# B&R Automation Studio project PickNPlaceD5Demo
Automation Studio 6.0.2.177; technology packages: mappCockpit 6.0.0, mappMotion 6.2.0, mappView 6.0.0, OpcUaCs 6.0.0

## Configuration Config1

### Task classes (Cpu.sw)
```
Cyclic#1 (cycle 2000 us, tolerance 0 us):
  APP_ConOut <- Conveyor.APP_ConveyorOut.prg
  APP_ConIn <- Conveyor.APP_ConveyorIn.prg
  APP_Robot1 <- Robots.Robot1.APP_Robot1.prg
DataObjects: McAcpSys, Arnc0sys, Acp10sys
NcDataObjects: mcdrivelog, gmcipuc, gmciplog, gmcipfub, gmcipfun, gmciplsm, gmciplbr, gmcipmxd, gmcipvar, gmcipsys, gmcipiec, gmcipesm, gmcipusm, gmcipcsm, gmcipui, gmcipubr, gmcipcbr, gmcipcfg, gmcipus, gmcipmx, Cam
Binaries: udbdef, TCData, mvLoader, arsvcreg, arflatprv, mCoWebSc, McAcpDrv, McAcpSim, McProfGen, McMechSys, arcoal, ashwac, arconfig, asfw, ashwd, iomap, User, Role, sysconf, TraceConfi, Settings, Config_1, Hierarchy, Config, AxisAx_1, Config_9, ComRobot, Config_7, Config_8, Config_6, ToolX20, AxesAxX21, GRobot1, GFRobot1, ARobot1, ComRobot1, WorkRobot1, GRobot2, MRobot1, GFRobot2, FeatX21, TrkDevX21, TrkDevConv, AxisAxX25, MecX20, AxesAxX20, WorkX20, FeatX20, DeltaX20, ComFeatX20, DeltaX21, TrkDevX20, vccddbox, vcfile, vccbtn, vcpdvnc, arialbd, vcmgr, vctcal, vcgclass, vcctext, vccnum, vcfntttf, vcdsloc, vccstr, arial, Visu03, vccshape, vcalarm, Visu01, vccdt, vccscale, vcchtml, vcchspot, vccbmp, vccpopup, vcshared, vcxml, vccurl, vcrt, vccslider, Visu02, vcnet, vcclbox, vcbclass, vcdsint, vcpdsw, vccovl, vccline, TCLang, visvc, vccdbox, vcpfar00, vcpfmtcx, vcpfapc, GrpMaster, Users, UsersLogin, TC, Files, DiagWebXs, AlmMaster, AlmHisMain, AlmMain, GrpVMaster, AlmVMaster, CfgPureVir, AxisPS, AxisAxXX1, AxisAxXX2, AxisMaster, MDevXX1, AxVMaster, GrpDevXX1, AlmDevXX1, GrPDevXX4, AlmDevXX4, GrPDevX10, AlmDevX10, AlmDevX20, GrpDevX20, AlmDevX21, GrpDevX21, AlmMBelts, GrpMBelts, AlmDevXX6, GrpDevXX6, AxesVAxX20, vcpfx20, AxisMBelts, MasMBelts, MBeltsPt, AxesVAxX25, AxesAxX10, AxesAxX25, WorkX10, CncXX6, MecX10, AxesVAxX10, DeltaX10, FeatXX6, FeatX10, ToolX10, ToolXX6, MecXX6, MotMaster, MotVMaster, vcctrend, MotDevX10, GrPDevXX3, AlmDevXX3, MotDevXX3, GrPDevXX2, MotDevXX1, AlmDevXX2, MotDevXX2, vcpkat, arnc0cfg, Sdc10map, Arnc0map, Sdc10map1, Sdc10map2, MotDevX20, MotDevX11, MotDevXX9, GrpDevXX9, AlmDevXX9, PML, MotDevXX6, CncDevXX6, MotDevXX7, AlmDevXX7, GrpDevXX7, Robot, AlmDevXX8, GrpDevXX8, MotSim, MotSpindle, MotDevXXA, AlmDevXXA, GrpDevXXA, GrpDevX11, AlmDevX11, OpcUaBasic, User_1, OpcUaMap, AlmHmi, AlmHistHmi, Groups, vccpiech, MotMac, acp10cfg, Acp10map
Libraries: standard, AsBrStr, sys_lib, runtime, AsArSdm, astime, brsystem, FileIO, AsIODiag, DataObj, AsArProf, AsMem, AsIOAcc, AsEPL, ASMcDcs, AsBrMath, visapi, ArTextSys, AsSem, AsIecCon, AsZip, powerlnk, aruser, asusb, ashw, arcert, arssl, aseth, asio, asarlog, vcresman, IecCheck, areventlog, MpRecipe, MpUserX, MpFile, MpAlarmX, MpCom, CoTrace, MpServer, McBase, MpBase, MpAxis, McAcpAx, McPathGen, McPureVAx, McAxGroup, McAxis, McProgInt, McTrkPath, McDS402Ax, MpRobotics, MpCnc, MpTool
```

### Hardware
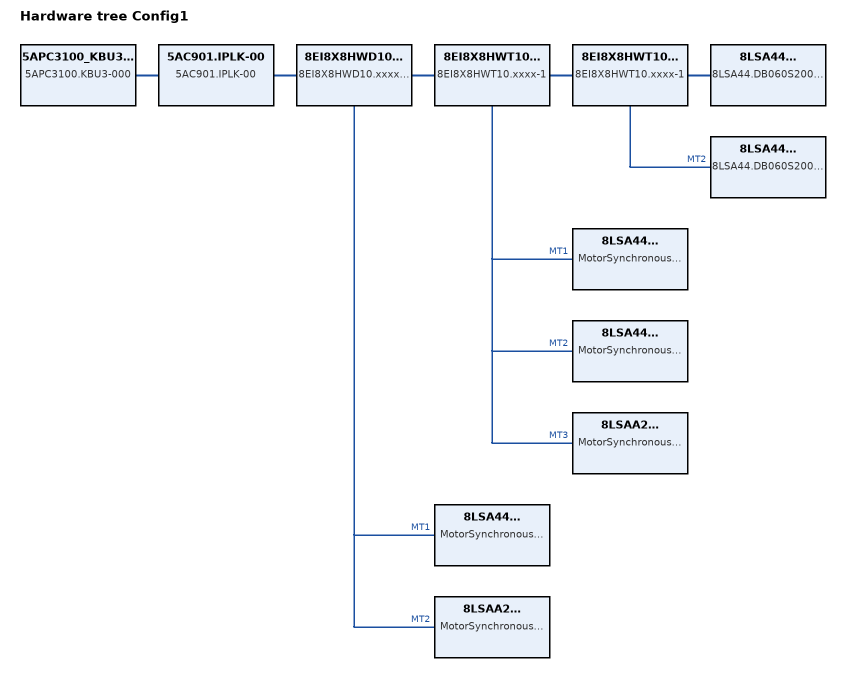
```
5AC901.IPLK-00 : 5AC901.IPLK-00 v2.0.0.0  [SL -> 5APC3100_KBU3_000.SL2]
  Connector IF1:
    DNAConfiguration = manual
    Channel1
    ChannelID1 = McAcpBroadcast
    ChannelType1 = OCTET[96]
5APC3100_KBU3_000 : 5APC3100.KBU3-000 v2.2.7.0
  Connector IF3:
    AssignedOperatingSystem = ARemb
    ActivateDevice = 1
    HostName = apc3100robert
    Mode = Manual
    InternetAddress = 10.43.51.43
    SubnetMask = 255.255.255.0
    Vnc1
    VncKeyMappingFile1 = 
    VncRefreshRate1 = 100
    ActivateSnmp = 2
  Connector IF4:
    AssignedOperatingSystem = ARemb
    ActivateDevice = 1
    HostName = apc3100robert
    Mode = DHCP Server
    InternetAddress = 192.168.20.254
    SubnetMask = 255.255.255.0
    Lease1
    LeaseName1 = Range1
    LeaseStartAddress1 = 192.168.20.100
    LeaseStopAddress1 = 192.168.20.110
    LeaseSubnetMask1 = 255.255.255.0
    Vnc1
    VncTitle1 = VNC
    ActivateSnmp = 2
  Connector IF5:
    AssignedOperatingSystem = ARemb
  Connector IF6:
    AssignedOperatingSystem = ARemb
  Connector IF7:
    AssignedOperatingSystem = ARemb
  Connector IF8:
    AssignedOperatingSystem = ARemb
  ConfigurationID = Template_X20CP1586
  UserPartitionSize = 5
  Simulation = 1
  TimerDeviceType = EPLX2X
  TimerDevice = 5AC901.IPLK-00.IF1
  IdleTaskClass = 4
  TaskClassIdleTime = 4000
  Cyclic1Duration = 2000
  Cyclic1Tolerance = 0
  Cyclic1Stack = 16384
  Cyclic2Duration = 4000
  Cyclic2Tolerance = 0
  Cyclic3Duration = 10000
  Cyclic3Tolerance = 0
  Cyclic4Duration = 20000
  Cyclic4Tolerance = 0
  Cyclic5Duration = 50000
  Cyclic5Tolerance = 0
  Cyclic6Duration = 100000
  Cyclic6Tolerance = 0
  Cyclic7Duration = 200000
  Cyclic7Tolerance = 0
  FileDevice1
  FileDeviceName1 = SceneViewer
  FileDevicePath1 = USER_PATH\..\..\..\..\..\FileDevices\SceneViewer
  FileDevice2
  FileDeviceName2 = CNC_PrgDir
  FileDevicePath2 = USER_PATH\..\..\..\..\..\FileDevices\GCode
  FileDevice3
  FileDeviceName3 = MPLogDir
  FileDevicePath3 = USER_PATH\..\..\..\..\..\FileDevices\Log
  FileDevice4
  FileDeviceName4 = DebugData
  FileDevicePath4 = USER_PATH\..\..\..\..\..\FileDevices\Debug
  EthernetDefaultGateway = 10.43.51.1
  ActivateFtpServer = 1
  FTPProtocol = 2
  FtpUser1
  FtpUsername1 = gmctest
  FtpUserPassword1 = dJg12F/7hd2fGO/QauVo5qNTeUud8LRwkPqca2btE1Q=
  FtpUserSalt1 = iGhlfz5v
  FTPAccessRight1 = 0
  FTPdevice1 = ALL
  ActivateWebServer = 1
  ActivateSdm = 1
8EI8X8HWD10.xxxx-1b_D5r1100R_1 : 8EI8X8HWD10.xxxx-1 v2.3.2.0 (NodeNumber=1)  [PLK1 -> 5AC901.IPLK-00.IF1 [Cable Type=PowerlinkCable, Length=10, Version=1.0.0.3]; PLK2 -> 8EI8X8HWT10.xxxx-1a_D5r1100R_1.PLK1 [Cable Type=PowerlinkCable, Length=10, Version=1.0.0.3]; MT2 -> 8LSAA2.D9045S200-3e_D5r1100R_1.MT]
  DriveConfiguration/Encoder/EncoderX41:
    InterfaceType = EnDat
  DriveConfiguration/Encoder/EncoderX42:
    InterfaceType = EnDat
  DriveConfiguration/Channel[1]/RealAxis:
    AxisReference = gAxisQ3_D5r1100R_1
  DriveConfiguration/Channel[1]/RealAxis/MechanicalElements/Gearbox:
    Input = 10
  DriveConfiguration/Channel[1]/RealAxis/EncoderLink:
    MotorAndPositionEncoder = EncoderX42
  DriveConfiguration/Channel[1]/RealAxis/Controller:
    Mode = PositionControllerWithTorqueFeedForward
  DriveConfiguration/Channel[1]/RealAxis/Controller/Mode/Position:
    ProportionalGain = 1.25
  DriveConfiguration/Channel[1]/RealAxis/Controller/Mode/Speed:
    ProportionalGain = 10.0
  DriveConfiguration/Channel[1]/RealAxis/Controller/Mode:
    FeedForward = CyclicValueFromAxesGroup
  DriveConfiguration/Channel[1]/RealAxis/Homing:
    Mode = Absolute
    RestorePositionVariable = 
  DriveConfiguration/Channel[1]/RealAxis/StopReaction:
    DriveError = CyclicDecelerationFromAxesGroup
  DriveConfiguration/Channel[1]/RealAxis/MovementErrorLimits:
    PositionError = 0.5
  DriveConfiguration/Channel[1]/RealAxis:
    JerkFilter = Used
  DriveConfiguration/Channel[1]/RealAxis/JerkFilter:
    JerkTime = 0.09
  DriveConfiguration/Channel[1]/RealAxis/DigitalInputs/HomingSwitch:
    Source = X8Trigger2
  DriveConfiguration/Channel[2]/RealAxis:
    AxisReference = gAxisQ5_D5r1100R_1
  DriveConfiguration/Channel[2]/RealAxis/MechanicalElements/Gearbox:
    Input = 10
  DriveConfiguration/Channel[2]/RealAxis/Controller:
    Mode = PositionControllerWithTorqueFeedForward
  DriveConfiguration/Channel[2]/RealAxis/Controller/Mode/Position:
    ProportionalGain = 25
  DriveConfiguration/Channel[2]/RealAxis/Controller/Mode/Speed:
    ProportionalGain = 1.25
  DriveConfiguration/Channel[2]/RealAxis/Controller/Mode:
    FeedForward = CyclicValueFromAxesGroup
  DriveConfiguration/Channel[2]/RealAxis/Homing:
    Mode = Absolute
    RestorePositionVariable = 
  DriveConfiguration/Channel[2]/RealAxis/StopReaction:
    DriveError = CyclicDecelerationFromAxesGroup
  DriveConfiguration/Channel[2]/RealAxis/MovementErrorLimits:
    PositionError = 0.5
  DriveConfiguration/Channel[2]/RealAxis:
    JerkFilter = Used
  DriveConfiguration/Channel[2]/RealAxis/JerkFilter:
    JerkTime = 0.09
8EI8X8HWT10.xxxx-1 : 8EI8X8HWT10.xxxx-1 v2.3.2.0 (NodeNumber=3)  [PLK1 -> 8EI8X8HWT10.xxxx-1a_D5r1100R_1.PLK2 [Cable Type=PowerlinkCable, Length=10, Version=1.0.0.3]; MT2 -> 8LSA44.DB060S200-3a.MT]
  DriveConfiguration/Module:
    McAcoposTypeID = AcoposP3TConfig
    ActivateACOPOSSimulationOnPLC = 0
    PowerSupply = AC
  DriveConfiguration/Encoder/EncoderX41:
    InterfaceType = NotUsed
  DriveConfiguration/Encoder/EncoderX42:
    InterfaceType = NotUsed
  DriveConfiguration/Encoder/EncoderX43:
    InterfaceType = NotUsed
  DriveConfiguration/Channel[1]/RealAxis:
    AxisReference = AxConveyorIn
    MechanicalElementsIsInvisible = 0
  DriveConfiguration/Channel[1]/RealAxis/MechanicalElements/Gearbox:
    InputIsReadOnly = 0
    Input = 1
    OutputIsReadOnly = 0
    Output = 1
  DriveConfiguration/Channel[1]/RealAxis/MechanicalElements/RotaryToLinearTransformation:
    ReferenceDistanceIsReadOnly = 0
    ReferenceDistance = 1
  DriveConfiguration/Channel[1]/RealAxis:
    EncoderLink = OneEncoder
  DriveConfiguration/Channel[1]/RealAxis/Controller:
    ModeIsReadOnly = 0
    Mode = PositionController
  DriveConfiguration/Channel[1]/RealAxis/Homing:
    ModeIsReadOnly = 0
    Mode = Direct
    RestorePositionVariable = 
  DriveConfiguration/Channel[1]/RealAxis/StopReaction:
    QuickstopIsReadOnly = 0
    Quickstop = DecelerationLimit
    DriveErrorIsReadOnly = 0
    DriveError = DecelerationLimit
  DriveConfiguration/Channel[1]/RealAxis/MovementErrorLimits:
    PositionError = 1.0
    VelocityErrorMonitoring = Automatic1
  DriveConfiguration/Channel[1]/RealAxis:
    JerkFilterIsReadOnly = 0
    JerkFilter = NotUsed
    ZeroVibrationFilter = NotUsed
  DriveConfiguration/Channel[1]/RealAxis/DigitalInputs/HomingSwitch:
    SourceIsReadOnly = 0
    Source = NotUsed
    Level = High
  DriveConfiguration/Channel[1]/RealAxis/DigitalInputs/PositiveLimitSwitch:
    SourceIsReadOnly = 0
    Source = NotUsed
    Level = High
  DriveConfiguration/Channel[1]/RealAxis/DigitalInputs/NegativeLimitSwitch:
    SourceIsReadOnly = 0
    Source = NotUsed
    Level = High
  DriveConfiguration/Channel[1]/RealAxis/DigitalInputs/Trigger1:
    Source = X8Trigger1
    Level = High
  DriveConfiguration/Channel[1]/RealAxis/DigitalInputs/Trigger2:
    Source = X8Trigger2
    Level = High
  DriveConfiguration/Channel[1]/RealAxis/DigitalInputs/Quickstop:
    Input = Trigger2
  DriveConfiguration/Channel[1]/RealAxis/Simulation:
    SimulationModeOnPLC = SetValueGeneration
    SimulationModeOnACOPOS = NotUsed
  DriveConfiguration/Channel[1]:
    VirtualAxis = NotUsed
    ExternalEncoderAxis = NotUsed
  DriveConfiguration/Channel[2]/RealAxis:
    AxisReference = AxConveyorOut
    MechanicalElementsIsInvisible = 0
  DriveConfiguration/Channel[2]/RealAxis/MechanicalElements/Gearbox:
    InputIsReadOnly = 0
    Input = 1
    OutputIsReadOnly = 0
    Output = 1
  DriveConfiguration/Channel[2]/RealAxis/MechanicalElements/RotaryToLinearTransformation:
    ReferenceDistanceIsReadOnly = 0
    ReferenceDistance = 1
  DriveConfiguration/Channel[2]/RealAxis:
    EncoderLink = OneEncoder
  DriveConfiguration/Channel[2]/RealAxis/Controller:
    ModeIsReadOnly = 0
    Mode = PositionController
  DriveConfiguration/Channel[2]/RealAxis/Homing:
    ModeIsReadOnly = 0
    Mode = Direct
    RestorePositionVariable = 
  DriveConfiguration/Channel[2]/RealAxis/StopReaction:
    QuickstopIsReadOnly = 0
    Quickstop = DecelerationLimit
    DriveErrorIsReadOnly = 0
    DriveError = DecelerationLimit
  DriveConfiguration/Channel[2]/RealAxis/MovementErrorLimits:
    PositionError = 1.0
    VelocityErrorMonitoring = Automatic1
  DriveConfiguration/Channel[2]/RealAxis:
    JerkFilterIsReadOnly = 0
    JerkFilter = NotUsed
    ZeroVibrationFilter = NotUsed
  DriveConfiguration/Channel[2]/RealAxis/DigitalInputs/HomingSwitch:
    SourceIsReadOnly = 0
    Source = NotUsed
    Level = High
  DriveConfiguration/Channel[2]/RealAxis/DigitalInputs/PositiveLimitSwitch:
    SourceIsReadOnly = 0
    Source = NotUsed
    Level = High
  DriveConfiguration/Channel[2]/RealAxis/DigitalInputs/NegativeLimitSwitch:
    SourceIsReadOnly = 0
    Source = NotUsed
    Level = High
  DriveConfiguration/Channel[2]/RealAxis/DigitalInputs/Trigger1:
    Source = X8Trigger1
    Level = High
  DriveConfiguration/Channel[2]/RealAxis/DigitalInputs/Trigger2:
    Source = X8Trigger2
    Level = High
  DriveConfiguration/Channel[2]/RealAxis/DigitalInputs/Quickstop:
    Input = Trigger2
  DriveConfiguration/Channel[2]/RealAxis/Simulation:
    SimulationModeOnPLC = SetValueGeneration
    SimulationModeOnACOPOS = NotUsed
  DriveConfiguration/Channel[2]/RealAxis/AxisFeatures:
    FeatureRef[1] = AxProfGenJerkLim
  DriveConfiguration/Channel[2]:
    VirtualAxis = NotUsed
    ExternalEncoderAxis = NotUsed
  DriveConfiguration/Channel[3]/RealAxis:
    AxisReference = 
    MechanicalElementsIsInvisible = 0
  DriveConfiguration/Channel[3]/RealAxis/MechanicalElements/Gearbox:
    InputIsReadOnly = 0
    Input = 1
    OutputIsReadOnly = 0
    Output = 1
  DriveConfiguration/Channel[3]/RealAxis/MechanicalElements/RotaryToLinearTransformation:
    ReferenceDistanceIsReadOnly = 0
    ReferenceDistance = 1
  DriveConfiguration/Channel[3]/RealAxis:
    EncoderLink = OneEncoder
  DriveConfiguration/Channel[3]/RealAxis/Controller:
    ModeIsReadOnly = 0
    Mode = PositionController
  DriveConfiguration/Channel[3]/RealAxis/Homing:
    ModeIsReadOnly = 0
    Mode = Direct
    RestorePositionVariable = 
  DriveConfiguration/Channel[3]/RealAxis/StopReaction:
    QuickstopIsReadOnly = 0
    Quickstop = DecelerationLimit
    DriveErrorIsReadOnly = 0
    DriveError = DecelerationLimit
  DriveConfiguration/Channel[3]/RealAxis/MovementErrorLimits:
    PositionError = 1.0
    VelocityErrorMonitoring = Automatic1
  DriveConfiguration/Channel[3]/RealAxis:
    JerkFilterIsReadOnly = 0
    JerkFilter = Used
  DriveConfiguration/Channel[3]/RealAxis/JerkFilter:
    JerkTime = 0.09
  DriveConfiguration/Channel[3]/RealAxis:
    ZeroVibrationFilter = NotUsed
  DriveConfiguration/Channel[3]/RealAxis/DigitalInputs/HomingSwitch:
    SourceIsReadOnly = 0
    Source = NotUsed
    Level = High
  DriveConfiguration/Channel[3]/RealAxis/DigitalInputs/PositiveLimitSwitch:
    SourceIsReadOnly = 0
    Source = NotUsed
    Level = High
  DriveConfiguration/Channel[3]/RealAxis/DigitalInputs/NegativeLimitSwitch:
    SourceIsReadOnly = 0
    Source = NotUsed
    Level = High
  DriveConfiguration/Channel[3]/RealAxis/DigitalInputs/Trigger1:
    Source = X8Trigger1
    Level = High
  DriveConfiguration/Channel[3]/RealAxis/DigitalInputs/Trigger2:
    Source = X8Trigger2
    Level = High
  DriveConfiguration/Channel[3]/RealAxis/DigitalInputs/Quickstop:
    Input = Trigger2
  DriveConfiguration/Channel[3]/RealAxis/Simulation:
    SimulationModeOnPLC = SetValueGeneration
    SimulationModeOnACOPOS = NotUsed
  DriveConfiguration/Channel[3]:
    VirtualAxis = NotUsed
    ExternalEncoderAxis = NotUsed
8EI8X8HWT10.xxxx-1a_D5r1100R_1 : 8EI8X8HWT10.xxxx-1 v2.3.2.0 (NodeNumber=2)  [PLK1 -> 8EI8X8HWD10.xxxx-1b_D5r1100R_1.PLK2 [Cable Type=PowerlinkCable, Length=10, Version=1.0.0.3]; PLK2 -> 8EI8X8HWT10.xxxx-1.PLK1 [Cable Type=PowerlinkCable, Length=10, Version=1.0.0.3]; MT2 -> 8LSA44.DB060S200-3b_D5r1100R_1.MT; MT3 -> 8LSAA2.D9045S200-3d_D5r1100R_1.MT]
  DriveConfiguration/Encoder/EncoderX41:
    InterfaceType = EnDat
  DriveConfiguration/Encoder/EncoderX42:
    InterfaceType = EnDat
  DriveConfiguration/Encoder/EncoderX43:
    InterfaceType = EnDat
  DriveConfiguration/Channel[1]/RealAxis:
    AxisReference = gAxisQ1_D5r1100R_1
  DriveConfiguration/Channel[1]/RealAxis/MechanicalElements/Gearbox:
    Input = 28
  DriveConfiguration/Channel[1]/RealAxis/Controller:
    Mode = PositionControllerWithTorqueFeedForward
  DriveConfiguration/Channel[1]/RealAxis/Controller/Mode/Position:
    ProportionalGain = 25
  DriveConfiguration/Channel[1]/RealAxis/Controller/Mode/Speed:
    ProportionalGain = 10
  DriveConfiguration/Channel[1]/RealAxis/Controller/Mode:
    FeedForward = CyclicValueFromAxesGroup
  DriveConfiguration/Channel[1]/RealAxis/Homing:
    Mode = Absolute
    RestorePositionVariable = 
  DriveConfiguration/Channel[1]/RealAxis/StopReaction:
    DriveError = CyclicDecelerationFromAxesGroup
  DriveConfiguration/Channel[1]/RealAxis/MovementErrorLimits:
    PositionError = 0.5
  DriveConfiguration/Channel[1]/RealAxis:
    JerkFilter = Used
  DriveConfiguration/Channel[1]/RealAxis/JerkFilter:
    JerkTime = 0.09
  DriveConfiguration/Channel[2]/RealAxis:
    AxisReference = gAxisQ2_D5r1100R_1
  DriveConfiguration/Channel[2]/RealAxis/MechanicalElements/Gearbox:
    Input = 28
  DriveConfiguration/Channel[2]/RealAxis/Controller:
    Mode = PositionControllerWithTorqueFeedForward
  DriveConfiguration/Channel[2]/RealAxis/Controller/Mode/Position:
    ProportionalGain = 25
  DriveConfiguration/Channel[2]/RealAxis/Controller/Mode/Speed:
    ProportionalGain = 10
  DriveConfiguration/Channel[2]/RealAxis/Controller/Mode:
    FeedForward = CyclicValueFromAxesGroup
  DriveConfiguration/Channel[2]/RealAxis/Homing:
    Mode = Absolute
    RestorePositionVariable = 
  DriveConfiguration/Channel[2]/RealAxis/StopReaction:
    DriveError = CyclicDecelerationFromAxesGroup
  DriveConfiguration/Channel[2]/RealAxis/MovementErrorLimits:
    PositionError = 0.5
  DriveConfiguration/Channel[2]/RealAxis:
    JerkFilter = Used
  DriveConfiguration/Channel[2]/RealAxis/JerkFilter:
    JerkTime = 0.09
  DriveConfiguration/Channel[3]/RealAxis:
    AxisReference = gAxisQ4_D5r1100R_1
  DriveConfiguration/Channel[3]/RealAxis/MechanicalElements/Gearbox:
    Input = 10
  DriveConfiguration/Channel[3]/RealAxis/Controller:
    Mode = PositionControllerWithTorqueFeedForward
  DriveConfiguration/Channel[3]/RealAxis/Controller/Mode/Position:
    ProportionalGain = 350
  DriveConfiguration/Channel[3]/RealAxis/Controller/Mode/Speed:
    ProportionalGain = 0.75
  DriveConfiguration/Channel[3]/RealAxis/Controller/Mode:
    FeedForward = CyclicValueFromAxesGroup
  DriveConfiguration/Channel[3]/RealAxis/Homing:
    Mode = Absolute
    RestorePositionVariable = 
  DriveConfiguration/Channel[3]/RealAxis/StopReaction:
    DriveError = CyclicDecelerationFromAxesGroup
  DriveConfiguration/Channel[3]/RealAxis/MovementErrorLimits:
    PositionError = 0.5
  DriveConfiguration/Channel[3]/RealAxis:
    JerkFilter = Used
  DriveConfiguration/Channel[3]/RealAxis/JerkFilter:
    JerkTime = 0.09
8LSA44.DB060S200-3 : 8LSA44.DB060S200-3 v2.2.0.2  [MT -> 8EI8X8HWT10.xxxx-1.MT1]
  M1/MotorParameters:
    MOTOR_AMB_TEMP_RATED = 40
  M1/MotorParameters/TemperatureSensor:
    MOTOR_TEMPSENS_LIM = 130
8LSA44.DB060S200-3a : 8LSA44.DB060S200-3 v2.2.0.2  [MT -> 8EI8X8HWT10.xxxx-1.MT2]
  M1/MotorParameters:
    MOTOR_AMB_TEMP_RATED = 40
  M1/MotorParameters/TemperatureSensor:
    MOTOR_TEMPSENS_LIM = 130
8LSA44.DB060S200-3a_D5r1100R_1 : MotorSynchronous_any v2.2.1.0  [MT -> 8EI8X8HWT10.xxxx-1a_D5r1100R_1.MT1]
  M1IsInvisible = 0
  TypeIsReadOnly = 0
  M1/MotorParameters:
    MOTOR_POLEPAIRS = 5
    MOTOR_SPEED_RATED = 6000
    MOTOR_SPEED_MAX = 12000
    MOTOR_VOLTAGE_RATED = 400
    MOTOR_CURR_RATED = 3.7
    MOTOR_CURR_STALL = 7.4
    MOTOR_CURR_MAX = 43.8
    MOTOR_TORQ_RATED = 3
    MOTOR_TORQ_STALL = 6
    MOTOR_TORQ_MAX = 22.8
    MOTOR_VOLTAGE_CONST = 49.22
    MOTOR_TORQ_CONST = 0.81
    MOTOR_STATOR_RESISTANCE = 0.862
    MOTOR_STATOR_INDUCTANCE = 6.2
    MOTOR_INERTIA = 2.73
    MOTOR_AMB_TEMP_RATED = 40
    VoltageLimitation = Used
  M1/MotorParameters/VoltageLimitation:
    MOTOR_UDC_MAX = 1000
  M1/MotorParameters/EncoderMounting:
    Angle = StoredOnEncoder
  M1/MotorParameters/TemperatureSensor:
    MOTOR_TEMPSENS_LIM = 130
    TemperatureSensorInterface = EncoderConnectorDigital
    MOTOR_TEMPSENS_PAR1 = 30
    MOTOR_TEMPSENS_PAR2 = 254
    MOTOR_TEMPSENS_PAR3 = -29.72
    MOTOR_TEMPSENS_PAR4 = -4.58
    MOTOR_TEMPSENS_PAR5 = 20.33
    MOTOR_TEMPSENS_PAR6 = 45.18
    MOTOR_TEMPSENS_PAR7 = 69.96
    MOTOR_TEMPSENS_PAR8 = 94.71
    MOTOR_TEMPSENS_PAR9 = 119.6
    MOTOR_TEMPSENS_PAR10 = 149.11
  M1/MotorParameters/TemperatureModel:
    MOTOR_WIND_TEMP_MAX = 110
  M1/MotorParameters/TemperatureModel/Calculation:
    MOTOR_WIND_CROSS_SECT = 0.985
    PIDENT_THERM_TRIP_TIME = 
    MOTOR_TAU_THERM = 1800
  M1:
    Brake = Used
  M1/Brake:
    MOTOR_BRAKE_CURR_RATED = 0.83
    MOTOR_BRAKE_TORQ_RATED = 8
    MOTOR_BRAKE_ON_TIME = 0.038
    MOTOR_BRAKE_OFF_TIME = 0.055
    MOTOR_BRAKE_INERTIA = 0.69
  M1/Encoder:
    MOTOR_ENCOD_ATTR = 1
    MOTOR_ENCOD_INERTIA = 0.022
    TemperatureSensor = Used
  M1/Encoder/TemperatureSensor:
    MOTOR_ENCOD_TEMP_LIM = 129
  M1:
    Gearbox = UsedWithDynamicTorqueLimitation
  M1/Gearbox/GearRatio:
    InputIsReadOnly = 0
    Input = 28
    OutputIsReadOnly = 0
    Output = 1
  M1/Gearbox:
    MOTORGEAR_SPEED_MAX = 5000
    MOTORGEAR_TORQ_NOM = 126
    MOTORGEAR_TORQ_MAX = 126
    MOTORGEAR_INERTIA = 0.51
    MOTORGEAR_VISC_FRIC = 0.002
    MOTORGEAR_STAT_FRIC = 0.22
8LSA44.DB060S200-3b_D5r1100R_1 : MotorSynchronous_any v2.2.1.0  [MT -> 8EI8X8HWT10.xxxx-1a_D5r1100R_1.MT2]
  M1IsInvisible = 0
  TypeIsReadOnly = 0
  M1/MotorParameters:
    MOTOR_POLEPAIRS = 5
    MOTOR_SPEED_RATED = 6000
    MOTOR_SPEED_MAX = 12000
    MOTOR_VOLTAGE_RATED = 400
    MOTOR_CURR_RATED = 3.7
    MOTOR_CURR_STALL = 7.4
    MOTOR_CURR_MAX = 43.8
    MOTOR_TORQ_RATED = 3
    MOTOR_TORQ_STALL = 6
    MOTOR_TORQ_MAX = 22.8
    MOTOR_VOLTAGE_CONST = 49.22
    MOTOR_TORQ_CONST = 0.81
    MOTOR_STATOR_RESISTANCE = 0.862
    MOTOR_STATOR_INDUCTANCE = 6.2
    MOTOR_INERTIA = 2.73
    MOTOR_AMB_TEMP_RATED = 40
    VoltageLimitation = Used
  M1/MotorParameters/VoltageLimitation:
    MOTOR_UDC_MAX = 1000
  M1/MotorParameters/EncoderMounting:
    Angle = StoredOnEncoder
  M1/MotorParameters/TemperatureSensor:
    MOTOR_TEMPSENS_LIM = 130
    TemperatureSensorInterface = EncoderConnectorDigital
    MOTOR_TEMPSENS_PAR1 = 30
    MOTOR_TEMPSENS_PAR2 = 254
    MOTOR_TEMPSENS_PAR3 = -29.72
    MOTOR_TEMPSENS_PAR4 = -4.58
    MOTOR_TEMPSENS_PAR5 = 20.33
    MOTOR_TEMPSENS_PAR6 = 45.18
    MOTOR_TEMPSENS_PAR7 = 69.96
    MOTOR_TEMPSENS_PAR8 = 94.71
    MOTOR_TEMPSENS_PAR9 = 119.6
    MOTOR_TEMPSENS_PAR10 = 149.11
  M1/MotorParameters/TemperatureModel:
    MOTOR_WIND_TEMP_MAX = 110
  M1/MotorParameters/TemperatureModel/Calculation:
    MOTOR_WIND_CROSS_SECT = 0.985
    PIDENT_THERM_TRIP_TIME = 
    MOTOR_TAU_THERM = 1800
  M1:
    Brake = Used
  M1/Brake:
    MOTOR_BRAKE_CURR_RATED = 0.83
    MOTOR_BRAKE_TORQ_RATED = 8
    MOTOR_BRAKE_ON_TIME = 0.038
    MOTOR_BRAKE_OFF_TIME = 0.055
    MOTOR_BRAKE_INERTIA = 0.69
  M1/Encoder:
    MOTOR_ENCOD_ATTR = 1
    MOTOR_ENCOD_INERTIA = 0.022
    TemperatureSensor = Used
  M1/Encoder/TemperatureSensor:
    MOTOR_ENCOD_TEMP_LIM = 129
  M1:
    Gearbox = UsedWithDynamicTorqueLimitation
  M1/Gearbox/GearRatio:
    InputIsReadOnly = 0
    Input = 28
    OutputIsReadOnly = 0
    Output = 1
  M1/Gearbox:
    MOTORGEAR_SPEED_MAX = 5000
    MOTORGEAR_TORQ_NOM = 126
    MOTORGEAR_TORQ_MAX = 126
    MOTORGEAR_INERTIA = 0.51
    MOTORGEAR_VISC_FRIC = 0.002
    MOTORGEAR_STAT_FRIC = 0.22
8LSA44.DB060S200-3c_D5r1100R_1 : MotorSynchronous_any v2.2.1.0  [MT -> 8EI8X8HWD10.xxxx-1b_D5r1100R_1.MT1]
  M1IsInvisible = 0
  TypeIsReadOnly = 0
  M1/MotorParameters:
    MOTOR_POLEPAIRS = 5
    MOTOR_SPEED_RATED = 6000
    MOTOR_SPEED_MAX = 12000
    MOTOR_VOLTAGE_RATED = 400
    MOTOR_CURR_RATED = 3.7
    MOTOR_CURR_STALL = 7.4
    MOTOR_CURR_MAX = 43.8
    MOTOR_TORQ_RATED = 3
    MOTOR_TORQ_STALL = 6
    MOTOR_TORQ_MAX = 22.8
    MOTOR_VOLTAGE_CONST = 49.22
    MOTOR_TORQ_CONST = 0.81
    MOTOR_STATOR_RESISTANCE = 0.862
    MOTOR_STATOR_INDUCTANCE = 6.2
    MOTOR_INERTIA = 2.73
    MOTOR_AMB_TEMP_RATED = 40
    VoltageLimitation = Used
  M1/MotorParameters/VoltageLimitation:
    MOTOR_UDC_MAX = 1000
  M1/MotorParameters/EncoderMounting:
    Angle = StoredOnEncoder
  M1/MotorParameters/TemperatureSensor:
    MOTOR_TEMPSENS_LIM = 130
    TemperatureSensorInterface = EncoderConnectorDigital
    MOTOR_TEMPSENS_PAR1 = 30
    MOTOR_TEMPSENS_PAR2 = 254
    MOTOR_TEMPSENS_PAR3 = -29.72
    MOTOR_TEMPSENS_PAR4 = -4.58
    MOTOR_TEMPSENS_PAR5 = 20.33
    MOTOR_TEMPSENS_PAR6 = 45.18
    MOTOR_TEMPSENS_PAR7 = 69.96
    MOTOR_TEMPSENS_PAR8 = 94.71
    MOTOR_TEMPSENS_PAR9 = 119.6
    MOTOR_TEMPSENS_PAR10 = 149.11
  M1/MotorParameters/TemperatureModel:
    MOTOR_WIND_TEMP_MAX = 110
  M1/MotorParameters/TemperatureModel/Calculation:
    MOTOR_WIND_CROSS_SECT = 0.985
    PIDENT_THERM_TRIP_TIME = 
    MOTOR_TAU_THERM = 1800
  M1:
    Brake = Used
  M1/Brake:
    MOTOR_BRAKE_CURR_RATED = 0.83
    MOTOR_BRAKE_TORQ_RATED = 8
    MOTOR_BRAKE_ON_TIME = 0.038
    MOTOR_BRAKE_OFF_TIME = 0.055
    MOTOR_BRAKE_INERTIA = 0.69
  M1/Encoder:
    MOTOR_ENCOD_ATTR = 1
    MOTOR_ENCOD_INERTIA = 0.022
    TemperatureSensor = Used
  M1/Encoder/TemperatureSensor:
    MOTOR_ENCOD_TEMP_LIM = 129
  M1:
    Gearbox = UsedWithDynamicTorqueLimitation
  M1/Gearbox/GearRatio:
    InputIsReadOnly = 0
    Input = 28
    OutputIsReadOnly = 0
    Output = 1
  M1/Gearbox:
    MOTORGEAR_SPEED_MAX = 5000
    MOTORGEAR_TORQ_NOM = 126
    MOTORGEAR_TORQ_MAX = 126
    MOTORGEAR_INERTIA = 0.51
    MOTORGEAR_VISC_FRIC = 0.002
    MOTORGEAR_STAT_FRIC = 0.22
8LSAA2.D9045S200-3d_D5r1100R_1 : MotorSynchronous_any v2.2.1.0  [MT -> 8EI8X8HWT10.xxxx-1a_D5r1100R_1.MT3]
  M1IsInvisible = 0
  TypeIsReadOnly = 0
  M1/MotorParameters:
    MOTOR_POLEPAIRS = 5
    MOTOR_SPEED_RATED = 4500
    MOTOR_SPEED_MAX = 7000
    MOTOR_VOLTAGE_RATED = 400
    MOTOR_CURR_RATED = 1.31
    MOTOR_CURR_STALL = 1.42
    MOTOR_CURR_MAX = 6
    MOTOR_TORQ_RATED = 1.27
    MOTOR_TORQ_STALL = 1.4
    MOTOR_TORQ_MAX = 4.5
    MOTOR_VOLTAGE_CONST = 58.64
    MOTOR_TORQ_CONST = 0.97
    MOTOR_STATOR_RESISTANCE = 13.9
    MOTOR_STATOR_INDUCTANCE = 27
    MOTOR_INERTIA = 0.38
    MOTOR_AMB_TEMP_RATED = 40
    VoltageLimitation = Used
  M1/MotorParameters/VoltageLimitation:
    MOTOR_UDC_MAX = 1000
  M1/MotorParameters/EncoderMounting:
    Angle = StoredOnEncoder
  M1/MotorParameters/TemperatureSensor:
    MOTOR_TEMPSENS_LIM = 130
    TemperatureSensorInterface = EncoderConnectorDigital
    MOTOR_TEMPSENS_PAR1 = 30
    MOTOR_TEMPSENS_PAR2 = 254
    MOTOR_TEMPSENS_PAR3 = -29.72
    MOTOR_TEMPSENS_PAR4 = -4.58
    MOTOR_TEMPSENS_PAR5 = 20.33
    MOTOR_TEMPSENS_PAR6 = 45.18
    MOTOR_TEMPSENS_PAR7 = 69.96
    MOTOR_TEMPSENS_PAR8 = 94.71
    MOTOR_TEMPSENS_PAR9 = 119.6
    MOTOR_TEMPSENS_PAR10 = 149.11
  M1/MotorParameters/TemperatureModel:
    MOTOR_WIND_TEMP_MAX = 110
  M1/MotorParameters/TemperatureModel/Calculation:
    MOTOR_WIND_CROSS_SECT = 0.126
    MOTOR_TAU_THERM = 1860
  M1:
    Brake = Used
  M1/Brake:
    MOTOR_BRAKE_CURR_RATED = 0.56
    MOTOR_BRAKE_TORQ_RATED = 3.2
    MOTOR_BRAKE_ON_TIME = 0.01
    MOTOR_BRAKE_OFF_TIME = 0.06
    MOTOR_BRAKE_INERTIA = 0.38
  M1/Encoder:
    MOTOR_ENCOD_ATTR = 1
    MOTOR_ENCOD_INERTIA = 0.004
    TemperatureSensor = Used
  M1/Encoder/TemperatureSensor:
    MOTOR_ENCOD_TEMP_LIM = 124
  M1:
    Gearbox = UsedWithDynamicTorqueLimitation
  M1/Gearbox/GearRatio:
    InputIsReadOnly = 0
    Input = 10
    OutputIsReadOnly = 0
    Output = 1
  M1/Gearbox:
    MOTORGEAR_SPEED_MAX = 7500
    MOTORGEAR_TORQ_NOM = 7
    MOTORGEAR_TORQ_MAX = 7
    MOTORGEAR_INERTIA = 0.16
    MOTORGEAR_VISC_FRIC = 0.01
    MOTORGEAR_STAT_FRIC = 0.1
8LSAA2.D9045S200-3e_D5r1100R_1 : MotorSynchronous_any v2.2.1.0  [MT -> 8EI8X8HWD10.xxxx-1b_D5r1100R_1.MT2]
  M1IsInvisible = 0
  TypeIsReadOnly = 0
  M1/MotorParameters:
    MOTOR_POLEPAIRS = 5
    MOTOR_SPEED_RATED = 4500
    MOTOR_SPEED_MAX = 7000
    MOTOR_VOLTAGE_RATED = 400
    MOTOR_CURR_RATED = 1.31
    MOTOR_CURR_STALL = 1.42
    MOTOR_CURR_MAX = 6
    MOTOR_TORQ_RATED = 1.27
    MOTOR_TORQ_STALL = 1.4
    MOTOR_TORQ_MAX = 4.5
    MOTOR_VOLTAGE_CONST = 58.64
    MOTOR_TORQ_CONST = 0.97
    MOTOR_STATOR_RESISTANCE = 13.9
    MOTOR_STATOR_INDUCTANCE = 27
    MOTOR_INERTIA = 0.38
    MOTOR_AMB_TEMP_RATED = 40
    VoltageLimitation = Used
  M1/MotorParameters/VoltageLimitation:
    MOTOR_UDC_MAX = 1000
  M1/MotorParameters/EncoderMounting:
    Angle = StoredOnEncoder
  M1/MotorParameters/TemperatureSensor:
    MOTOR_TEMPSENS_LIM = 130
    TemperatureSensorInterface = EncoderConnectorDigital
    MOTOR_TEMPSENS_PAR1 = 30
    MOTOR_TEMPSENS_PAR2 = 254
    MOTOR_TEMPSENS_PAR3 = -29.72
    MOTOR_TEMPSENS_PAR4 = -4.58
    MOTOR_TEMPSENS_PAR5 = 20.33
    MOTOR_TEMPSENS_PAR6 = 45.18
    MOTOR_TEMPSENS_PAR7 = 69.96
    MOTOR_TEMPSENS_PAR8 = 94.71
    MOTOR_TEMPSENS_PAR9 = 119.6
    MOTOR_TEMPSENS_PAR10 = 149.11
  M1/MotorParameters/TemperatureModel:
    MOTOR_WIND_TEMP_MAX = 110
  M1/MotorParameters/TemperatureModel/Calculation:
    MOTOR_WIND_CROSS_SECT = 0.126
    MOTOR_TAU_THERM = 1860
  M1:
    Brake = Used
  M1/Brake:
    MOTOR_BRAKE_CURR_RATED = 0.56
    MOTOR_BRAKE_TORQ_RATED = 3.2
    MOTOR_BRAKE_ON_TIME = 0.01
    MOTOR_BRAKE_OFF_TIME = 0.06
    MOTOR_BRAKE_INERTIA = 0.38
  M1/Encoder:
    MOTOR_ENCOD_ATTR = 1
    MOTOR_ENCOD_INERTIA = 0.004
    TemperatureSensor = Used
  M1/Encoder/TemperatureSensor:
    MOTOR_ENCOD_TEMP_LIM = 124
  M1:
    Gearbox = UsedWithDynamicTorqueLimitation
  M1/Gearbox/GearRatio:
    InputIsReadOnly = 0
    Input = 10
    OutputIsReadOnly = 0
    Output = 1
  M1/Gearbox:
    MOTORGEAR_SPEED_MAX = 7500
    MOTORGEAR_TORQ_NOM = 7
    MOTORGEAR_TORQ_MAX = 7
    MOTORGEAR_INERTIA = 0.16
    MOTORGEAR_VISC_FRIC = 0.01
    MOTORGEAR_STAT_FRIC = 0.1
```

### Config_10.dynpartable - 5APC3100_KBU3_000/mappMotion/Codian_D5r1100R_1/Config_10.dynpartable
```
Element ProductLoad_2 (Type=dynpartable)
  Row[1]:
    Value = 1.0
    Unit = kg
    Description = Mass
  Row[2]:
    Index = 1
    Unit = m
    Description = Center of gravity - X direction
  Row[3]:
    Index = 2
    Unit = m
    Description = Center of gravity - Y direction
  Row[4]:
    Index = 3
    Unit = m
    Description = Center of gravity - Z direction
  Row[5]:
    Index = 4
    Unit = kg m^2
    Description = Moment of inertia about X
  Row[6]:
    Index = 5
    Unit = kg m^2
    Description = Moment of inertia about Y
  Row[7]:
    Index = 6
    Unit = kg m^2
    Description = Moment of inertia about Z
  Row[8]:
    Index = 1000
    Value = 1
    Unit = 
    Description = 0 (toolDynPar), 1 (productLoadPar)
```

### Config_11.tool - 5APC3100_KBU3_000/mappMotion/Codian_D5r1100R_1/Config_11.tool
```
Element Tool_1 (Type=tool)
```

### Config_4.dynpartable - 5APC3100_KBU3_000/mappMotion/Codian_D5r1100R_1/Config_4.dynpartable
```
Element ProductLoad_1 (Type=dynpartable)
  Row[1]:
    Value = 0.5
    Unit = kg
    Description = Mass
  Row[2]:
    Index = 1
    Unit = m
    Description = Center of gravity - X direction
  Row[3]:
    Index = 2
    Unit = m
    Description = Center of gravity - Y direction
  Row[4]:
    Index = 3
    Unit = m
    Description = Center of gravity - Z direction
  Row[5]:
    Index = 4
    Unit = kg m^2
    Description = Moment of inertia about X
  Row[6]:
    Index = 5
    Unit = kg m^2
    Description = Moment of inertia about Y
  Row[7]:
    Index = 6
    Unit = kg m^2
    Description = Moment of inertia about Z
  Row[8]:
    Index = 1000
    Value = 1
    Unit = 
    Description = 0 (toolDynPar), 1 (productLoadPar)
```

### Config_5.tooltable - 5APC3100_KBU3_000/mappMotion/Codian_D5r1100R_1/Config_5.tooltable
```
Element ToolTable_1 (Type=tooltable)
  Row[1]:
    Index = 3
    ToolDataRef = Tool_1
    ToolDynParDataRef = 
  Row[2]:
    ToolDynParDataRef = ProductLoad_1
  Row[3]:
    Index = 2
    ToolDynParDataRef = ProductLoad_2
```

### Config_6.axesgroup - 5APC3100_KBU3_000/mappMotion/Codian_D5r1100R_1/Config_6.axesgroup
```
Element gAxesGroup_D5r1100R_1 (Type=axesgroup)
  Type = PathGenAxesGroup
    ProcessingTaskClass = 1
    PhysicalAxes:
      JointAxes:
        JointAxis[1]:
          AxisRef = gAxisQ1_D5r1100R_1
        JointAxis[2]:
          AxisRef = gAxisQ2_D5r1100R_1
        JointAxis[3]:
          AxisRef = gAxisQ3_D5r1100R_1
        JointAxis[4]:
          Name = QC
          AxisRef = gAxisQ4_D5r1100R_1
        JointAxis[5]:
          Name = QA
          AxisRef = gAxisQ5_D5r1100R_1
    MechanicalSystem:
      MechSysRef = MechSys_D5r1100R_1
    BasicSettings:
      GeometryPlanning:
        MaxTangentialTransitionDeviation = 0.05
      TrajectoryPlanning:
        LimitCheckResolution:
          Time = 0.005
        BufferTime:
          Time = 0.05
      Miscellaneous:
        TimeStretchOverride:
          JerkSuppression = Basic
            AdaptationTime = 0.3
    StopReaction:
      AxisError:
        AxisReactionIsReadOnly = 1
        AxisReaction = DynamicStop
          ModeIsReadOnly = 1
    AxesGroupFeatures:
      FeatureRef[1] = Feature_Programs_D5r1100R_1
      FeatureRef[2] = Feature_FrameHierachy
      FeatureRef[3] = Feature_InterpreterLog
      FeatureRef[4] = Feature_MFunctions
      FeatureRef[5] = Feature_Monitoring
      FeatureRef[6] = Feature_PathDefRobot
      FeatureRef[7] = Feature_TrackingRobot
      FeatureRef[8] = Feature_WorkspaceMonitoring
      FeatureRef[9] = Feature_Signaling
      FeatureRef[10] = Feature_Tool
```

### Config_7.axis - 5APC3100_KBU3_000/mappMotion/Codian_D5r1100R_1/Config_7.axis
```
Element gAxisQ1_D5r1100R_1 (Type=axis)
  BaseTypeIsReadOnly = 0
  BaseType = RotaryBounded
    MeasurementUnitIsReadOnly = 1
    MeasurementUnit = 17476
    MeasurementResolutionIsReadOnly = 1
    MeasurementResolution = 0.001
    CountDirectionIsReadOnly = 1
    CountDirection = Inverse
  MovementLimitsIsReadOnly = 0
  MovementLimits = InternalForPathControlledAxis
    Position:
      LowerLimitMin = -47
      UpperLimitMax = 99.5
      LowerLimit = -47
      UpperLimit = 99.5
    VelocityIsReadOnly = 0
    Velocity:
      VelocityMax = 3.4E38
      Velocity = 1160
    AccelerationIsReadOnly = 0
    Acceleration:
      AccelerationMax = 3.4E38
      Acceleration = 35000
    DecelerationIsReadOnly = 0
    Deceleration:
      DecelerationMax = 3.4E38
      Deceleration = 35000
    JerkIsReadOnly = 0
    Jerk = Advanced
      JerkAccelerationPositiveMin = 0
      JerkAccelerationPositiveMax = 3.4E38
      JerkAccelerationPositive = 1500000
      JerkAccelerationNegativeMin = 0
      JerkAccelerationNegativeMax = 3.4E38
      JerkAccelerationNegative = 1500000
      JerkDecelerationPositiveMin = 0
      JerkDecelerationPositiveMax = 3.4E38
      JerkDecelerationPositive = 1500000
      JerkDecelerationNegativeMin = 0
      JerkDecelerationNegativeMax = 3.4E38
      JerkDecelerationNegative = 1500000
    TorqueIsInvisible = 0
    TorqueIsReadOnly = 0
    Torque = Basic
      TorqueMax = 3.4E38
      Torque = 11
  Alarms = None
Element gAxisQ2_D5r1100R_1 (Type=axis)
  BaseTypeIsReadOnly = 0
  BaseType = RotaryBounded
    MeasurementUnitIsReadOnly = 1
    MeasurementUnit = 17476
    MeasurementResolutionIsReadOnly = 1
    MeasurementResolution = 0.001
    CountDirectionIsReadOnly = 1
    CountDirection = Inverse
  MovementLimitsIsReadOnly = 0
  MovementLimits = InternalForPathControlledAxis
    Position:
      LowerLimitMin = -47
      UpperLimitMax = 99.5
      LowerLimit = -47
      UpperLimit = 99.5
    VelocityIsReadOnly = 0
    Velocity:
      VelocityMax = 3.4E38
      Velocity = 1160
    AccelerationIsReadOnly = 0
    Acceleration:
      AccelerationMax = 3.4E38
      Acceleration = 35000
    DecelerationIsReadOnly = 0
    Deceleration:
      DecelerationMax = 3.4E38
      Deceleration = 35000
    JerkIsReadOnly = 0
    Jerk = Advanced
      JerkAccelerationPositiveMin = 0
      JerkAccelerationPositiveMax = 3.4E38
      JerkAccelerationPositive = 1500000
      JerkAccelerationNegativeMin = 0
      JerkAccelerationNegativeMax = 3.4E38
      JerkAccelerationNegative = 1500000
      JerkDecelerationPositiveMin = 0
      JerkDecelerationPositiveMax = 3.4E38
      JerkDecelerationPositive = 1500000
      JerkDecelerationNegativeMin = 0
      JerkDecelerationNegativeMax = 3.4E38
      JerkDecelerationNegative = 1500000
    TorqueIsInvisible = 0
    TorqueIsReadOnly = 0
    Torque = Basic
      TorqueMax = 3.4E38
      Torque = 11
  Alarms = None
Element gAxisQ3_D5r1100R_1 (Type=axis)
  BaseTypeIsReadOnly = 0
  BaseType = RotaryBounded
    MeasurementUnitIsReadOnly = 1
    MeasurementUnit = 17476
    MeasurementResolutionIsReadOnly = 1
    MeasurementResolution = 0.001
    CountDirectionIsReadOnly = 1
    CountDirection = Inverse
  MovementLimitsIsReadOnly = 0
  MovementLimits = InternalForPathControlledAxis
    Position:
      LowerLimitMin = -47
      UpperLimitMax = 99.5
      LowerLimit = -47
      UpperLimit = 99.5
    VelocityIsReadOnly = 0
    Velocity:
      VelocityMax = 3.4E38
      Velocity = 1160
    AccelerationIsReadOnly = 0
    Acceleration:
      AccelerationMax = 3.4E38
      Acceleration = 35000
    DecelerationIsReadOnly = 0
    Deceleration:
      DecelerationMax = 3.4E38
      Deceleration = 35000
    JerkIsReadOnly = 0
    Jerk = Advanced
      JerkAccelerationPositiveMin = 0
      JerkAccelerationPositiveMax = 3.4E38
      JerkAccelerationPositive = 1500000
      JerkAccelerationNegativeMin = 0
      JerkAccelerationNegativeMax = 3.4E38
      JerkAccelerationNegative = 1500000
      JerkDecelerationPositiveMin = 0
      JerkDecelerationPositiveMax = 3.4E38
      JerkDecelerationPositive = 1500000
      JerkDecelerationNegativeMin = 0
      JerkDecelerationNegativeMax = 3.4E38
      JerkDecelerationNegative = 1500000
    TorqueIsInvisible = 0
    TorqueIsReadOnly = 0
    Torque = Basic
      TorqueMax = 3.4E38
      Torque = 11
  Alarms = None
Element gAxisQ4_D5r1100R_1 (Type=axis)
  BaseTypeIsReadOnly = 0
  BaseType = Rotary
    MeasurementUnitIsReadOnly = 1
    MeasurementUnit = 17476
    MeasurementResolutionIsReadOnly = 1
    MeasurementResolution = 0.001
    CountDirectionIsReadOnly = 1
    CountDirection = Standard
  MovementLimitsIsReadOnly = 0
  MovementLimits = InternalForPathControlledAxis
    Position:
      LowerLimitMin = -1000.0
      UpperLimitMax = 1000.0
      LowerLimit = -1000.0
      UpperLimit = 1000.0
    VelocityIsReadOnly = 0
    Velocity:
      VelocityMax = 3.4E38
      Velocity = 3600
    AccelerationIsReadOnly = 0
    Acceleration:
      AccelerationMax = 3.4E38
      Acceleration = 100000
    DecelerationIsReadOnly = 0
    Deceleration:
      DecelerationMax = 3.4E38
      Deceleration = 100000
    JerkIsReadOnly = 0
    Jerk = Advanced
      JerkAccelerationPositiveMin = 0
      JerkAccelerationPositiveMax = 3.4E38
      JerkAccelerationPositive = 6000000
      JerkAccelerationNegativeMin = 0
      JerkAccelerationNegativeMax = 3.4E38
      JerkAccelerationNegative = 6000000
      JerkDecelerationPositiveMin = 0
      JerkDecelerationPositiveMax = 3.4E38
      JerkDecelerationPositive = 6000000
      JerkDecelerationNegativeMin = 0
      JerkDecelerationNegativeMax = 3.4E38
      JerkDecelerationNegative = 6000000
    TorqueIsInvisible = 0
    TorqueIsReadOnly = 0
    Torque = Basic
      TorqueMax = 3.4E38
      Torque = 1.2
  Alarms = None
Element gAxisQ5_D5r1100R_1 (Type=axis)
  BaseTypeIsReadOnly = 0
  BaseType = Rotary
    MeasurementUnitIsReadOnly = 1
    MeasurementUnit = 17476
    MeasurementResolutionIsReadOnly = 1
    MeasurementResolution = 0.001
    CountDirectionIsReadOnly = 1
    CountDirection = Standard
  MovementLimitsIsReadOnly = 0
  MovementLimits = InternalForPathControlledAxis
    Position:
      LowerLimitMin = -186.01
      UpperLimitMax = 186.01
      LowerLimit = -186.01
      UpperLimit = 186.01
    VelocityIsReadOnly = 0
    Velocity:
      VelocityMax = 3.4E38
      Velocity = 3300
    AccelerationIsReadOnly = 0
    Acceleration:
      AccelerationMax = 3.4E38
      Acceleration = 100000
    DecelerationIsReadOnly = 0
    Deceleration:
      DecelerationMax = 3.4E38
      Deceleration = 100000
    JerkIsReadOnly = 0
    Jerk = Advanced
      JerkAccelerationPositiveMin = 0
      JerkAccelerationPositiveMax = 3.4E38
      JerkAccelerationPositive = 6000000
      JerkAccelerationNegativeMin = 0
      JerkAccelerationNegativeMax = 3.4E38
      JerkAccelerationNegative = 6000000
      JerkDecelerationPositiveMin = 0
      JerkDecelerationPositiveMax = 3.4E38
      JerkDecelerationPositive = 6000000
      JerkDecelerationNegativeMin = 0
      JerkDecelerationNegativeMax = 3.4E38
      JerkDecelerationNegative = 6000000
    TorqueIsInvisible = 0
    TorqueIsReadOnly = 0
    Torque = Basic
      TorqueMax = 3.4E38
      Torque = 2
  Alarms = None
```

### Config_8.mechanicalsystem - 5APC3100_KBU3_000/mappMotion/Codian_D5r1100R_1/Config_8.mechanicalsystem
```
Element MechSys_D5r1100R_1 (Type=mechanicalsystem)
  TypeIsReadOnly = 1
  Type = Delta
    SubtypeIsReadOnly = 1
    Subtype = 5AxesDeltaA
      SceneViewerObject = Generic
      DescriptionIsReadOnly = 1
      Description = Standard
        Dimensions:
          BasePlatform:
            CenterIsReadOnly = 0
            Center:
              X = 0.0
              Y = 0.0
              Z = 0
            ArmLinkPointIsReadOnly = 0
            Arm1LinkPoint:
              Angle = 0.0
              Radius = 200
              Z = -90
            Arm2LinkPoint:
              Angle = -120.0
              Radius = 200
              Z = -90
            Arm3LinkPoint:
              Angle = -240.0
              Radius = 200
              Z = -90
          Arms:
            ArmIsReadOnly = 0
            Arm1:
              UpperArmLength = 320
              LowerArmLength = 850
            Arm2:
              UpperArmLength = 320
              LowerArmLength = 850
            Arm3:
              UpperArmLength = 320
              LowerArmLength = 850
            LowerArmPairDistance = 104
          EndEffectorPlatform:
            ArmLinkPointIsReadOnly = 0
            Arm1LinkPoint:
              Radius = 66
              Z = 0.0
            Arm2LinkPoint:
              Radius = 66
              Z = 0.0
            Arm3LinkPoint:
              Radius = 66
              Z = 0.0
            TranslationToQCIsReadOnly = 0
            TranslationToQC:
              X = 27.5
              Y = 0.0
              Z = 0.0
            TranslationFromQCToQAIsReadOnly = 0
            TranslationFromQCToQA:
              X = 0.0
              Y = 0.0
              Z = -74.9
            TranslationFromQAToFlangeIsReadOnly = 0
            TranslationFromQAToFlange:
              X = 0.0
              Y = 0.0
              Z = -80
        Offsets:
          JointAxisIsReadOnly = 0
          JointAxis[1] = 0.0
          JointAxis[2] = 0.0
          JointAxis[3] = 0.0
          JointAxis[4] = 0.0
          JointAxis[5] = 0.0
        CountDirections:
          JointAxisIsReadOnly = 0
          JointAxis[1] = Standard
          JointAxis[2] = Standard
          JointAxis[3] = Standard
          JointAxis[4] = Standard
          JointAxis[5] = Standard
      CoordinatesNames = Default
        XCoordinateName = X
        YCoordinateName = Y
        ZCoordinateName = Z
        CCoordinateName = C
        ACoordinateName = A
      TcpOrientation:
        Frames = Used
      WireFrameModelIsReadOnly = 0
      WireFrameModel = Standard
        UpperArm1IsReadOnly = 0
        UpperArm1 = ConnectionLine
          DistanceMin = -1.79769313486231E308
          DistanceMax = 1.79769313486231E308
          Distance = 5
        LowerArm1IsReadOnly = 0
        LowerArm1 = ConnectionLine
          DistanceMin = -1.79769313486231E308
          DistanceMax = 1.79769313486231E308
          Distance = 5
        UpperArm2IsReadOnly = 0
        UpperArm2 = ConnectionLine
          DistanceMin = -1.79769313486231E308
          DistanceMax = 1.79769313486231E308
          Distance = 5
        LowerArm2IsReadOnly = 0
        LowerArm2 = ConnectionLine
          DistanceMin = -1.79769313486231E308
          DistanceMax = 1.79769313486231E308
          Distance = 5
        UpperArm3IsReadOnly = 0
        UpperArm3 = ConnectionLine
          DistanceMin = -1.79769313486231E308
          DistanceMax = 1.79769313486231E308
          Distance = 5
        LowerArm3IsReadOnly = 0
        LowerArm3 = ConnectionLine
          DistanceMin = -1.79769313486231E308
          DistanceMax = 1.79769313486231E308
          Distance = 5
        EndEffectorPlatformToQCIsReadOnly = 0
        EndEffectorPlatformToQC = ConnectionLine
          DistanceMin = -1.79769313486231E308
          DistanceMax = 1.79769313486231E308
          Distance = 0.0
        QCToQAIsReadOnly = 0
        QCToQA = ConnectionLine
          DistanceMin = -1.79769313486231E308
          DistanceMax = 1.79769313486231E308
          Distance = 0.0
        QAToFlangeIsReadOnly = 0
        QAToFlange = ConnectionLine
          DistanceMin = -1.79769313486231E308
          DistanceMax = 1.79769313486231E308
          Distance = 0.0
        FlangeToTcp = NotUsed
      DynamicModelIsReadOnly = 0
      DynamicModel = DynParTable
        TableRef
      InternalDynamicModelIsReadOnly = 1
      InternalDynamicModel = Used
        TypeIsReadOnly = 1
        Type = D5-1100-S026-R100
        Row[1]:
          Index = 0
          Value = 3
          Unit = 
          Description = type of robot dyn par model
        Row[2]:
          Index = 1
          Value = 1.017
          Unit = kg
          Description = m1
        Row[3]:
          Index = 2
          Value = 0.1042425
          Unit = kgm
          Description = m1*rc1x
        Row[4]:
          Index = 3
          Value = 0
          Unit = kgm
          Description = m1*rc1y
        Row[5]:
          Index = 4
          Value = 0.0044748
          Unit = kgm
          Description = m1*rc1z
        Row[6]:
          Index = 5
          Value = 0
          Unit = kgm^2
          Description = m1*rc1x*rc1y
        Row[7]:
          Index = 6
          Value = 0
          Unit = kgm^2
          Description = m1*rc1y*rc1z
        Row[8]:
          Index = 7
          Value = 0.000458667
          Unit = kgm^2
          Description = m1*rc1x*rc1z
        Row[9]:
          Index = 8
          Value = 0.01068485625
          Unit = kgm^2
          Description = m1*rc1x^2
        Row[10]:
          Index = 9
          Value = 0
          Unit = kgm^2
          Description = m1*rc1y^2
        Row[11]:
          Index = 10
          Value = 0.00001968912
          Unit = kgm^2
          Description = m1*rc1z^2
        Row[12]:
          Index = 11
          Value = 0
          Unit = kgm^2
          Description = Jxx1
        Row[13]:
          Index = 12
          Value = 0.0129
          Unit = kgm^2
          Description = Jyy1
        Row[14]:
          Index = 13
          Value = 0
          Unit = kgm^2
          Description = Jzz1
        Row[15]:
          Index = 14
          Value = 1.017
          Unit = kg
          Description = m2
        Row[16]:
          Index = 15
          Value = 0.1042425
          Unit = kgm
          Description = m2*rc2x
        Row[17]:
          Index = 16
          Value = 0
          Unit = kgm
          Description = m2*rc2y
        Row[18]:
          Index = 17
          Value = 0.0044748
          Unit = kgm
          Description = m2*rc2z
        Row[19]:
          Index = 18
          Value = 0
          Unit = kgm^2
          Description = m2*rc2x*rc2y
        Row[20]:
          Index = 19
          Value = 0
          Unit = kgm^2
          Description = m2*rc2y*rc2z
        Row[21]:
          Index = 20
          Value = 0.000458667
          Unit = kgm^2
          Description = m2*rc2x*rc2z
        Row[22]:
          Index = 21
          Value = 0.01068485625
          Unit = kgm^2
          Description = m2*rc2x^2
        Row[23]:
          Index = 22
          Value = 0
          Unit = kgm^2
          Description = m2*rc2y^2
        Row[24]:
          Index = 23
          Value = 0.00001968912
          Unit = kgm^2
          Description = m2*rc2z^2
        Row[25]:
          Index = 24
          Value = 0
          Unit = kgm^2
          Description = Jxx2
        Row[26]:
          Index = 25
          Value = 0.0129
          Unit = kgm^2
          Description = Jyy2
        Row[27]:
          Index = 26
          Value = 0
          Unit = kgm^2
          Description = Jzz2
        Row[28]:
          Index = 27
          Value = 1.017
          Unit = kg
          Description = m3
        Row[29]:
          Index = 28
          Value = 0.1042425
          Unit = kgm
          Description = m3*rc3x
        Row[30]:
          Index = 29
          Value = 0
          Unit = kgm
          Description = m3*rc3y
        Row[31]:
          Index = 30
          Value = 0.0044748
          Unit = kgm
          Description = m3*rc3z
        Row[32]:
          Index = 31
          Value = 0
          Unit = kgm^2
          Description = m3*rc3x*rc3y
        Row[33]:
          Index = 32
          Value = 0
          Unit = kgm^2
          Description = m3*rc3y*rc3z
        Row[34]:
          Index = 33
          Value = 0.000458667
          Unit = kgm^2
          Description = m3*rc3x*rc3z
        Row[35]:
          Index = 34
          Value = 0.01068485625
          Unit = kgm^2
          Description = m3*rc3x^2
        Row[36]:
          Index = 35
          Value = 0
          Unit = kgm^2
          Description = m3*rc3y^2
        Row[37]:
          Index = 36
          Value = 0.00001968912
          Unit = kgm^2
          Description = m3*rc3z^2
        Row[38]:
          Index = 37
          Value = 0
          Unit = kgm^2
          Description = Jxx3
        Row[39]:
          Index = 38
          Value = 0.0129
          Unit = kgm^2
          Description = Jyy3
        Row[40]:
          Index = 39
          Value = 0
          Unit = kgm^2
          Description = Jzz3
        Row[41]:
          Index = 40
          Value = 0.394
          Unit = kg
          Description = m4
        Row[42]:
          Index = 41
          Value = 0
          Unit = kgm
          Description = m4*rc4x
        Row[43]:
          Index = 42
          Value = 0
          Unit = kgm
          Description = m4*rc4y
        Row[44]:
          Index = 43
          Value = 0.16745
          Unit = kgm
          Description = m4*rc4z
        Row[45]:
          Index = 44
          Value = 0
          Unit = kgm^2
          Description = m4*rc4x*rc4y
        Row[46]:
          Index = 45
          Value = 0
          Unit = kgm^2
          Description = m4*rc4y*rc4z
        Row[47]:
          Index = 46
          Value = 0
          Unit = kgm^2
          Description = m4*rc4x*rc4z
        Row[48]:
          Index = 47
          Value = 0
          Unit = kgm^2
          Description = m4*rc4x^2
        Row[49]:
          Index = 48
          Value = 0
          Unit = kgm^2
          Description = m4*rc4y^2
        Row[50]:
          Index = 49
          Value = 0.16745
          Unit = kgm^2
          Description = m4*rc4z^2
        Row[51]:
          Index = 50
          Value = 0.038
          Unit = kgm^2
          Description = Jxx4
        Row[52]:
          Index = 51
          Value = 0.038
          Unit = kgm^2
          Description = Jyy4
        Row[53]:
          Index = 52
          Value = 0
          Unit = kgm^2
          Description = Jzz4
        Row[54]:
          Index = 53
          Value = 0.394
          Unit = kg
          Description = m5
        Row[55]:
          Index = 54
          Value = 0
          Unit = kgm
          Description = m5*rc5x
        Row[56]:
          Index = 55
          Value = 0
          Unit = kgm
          Description = m5*rc5y
        Row[57]:
          Index = 56
          Value = 0.16745
          Unit = kgm
          Description = m5*rc5z
        Row[58]:
          Index = 57
          Value = 0
          Unit = kgm^2
          Description = m5*rc5x*rc5y
        Row[59]:
          Index = 58
          Value = 0
          Unit = kgm^2
          Description = m5*rc5y*rc5z
        Row[60]:
          Index = 59
          Value = 0
          Unit = kgm^2
          Description = m5*rc5x*rc5z
        Row[61]:
          Index = 60
          Value = 0
          Unit = kgm^2
          Description = m5*rc5x^2
        Row[62]:
          Index = 61
          Value = 0
          Unit = kgm^2
          Description = m5*rc5y^2
        Row[63]:
          Index = 62
          Value = 0.16745
          Unit = kgm^2
          Description = m5*rc5z^2
        Row[64]:
          Index = 63
          Value = 0.038
          Unit = kgm^2
          Description = Jxx5
        Row[65]:
          Index = 64
          Value = 0.038
          Unit = kgm^2
          Description = Jyy5
        Row[66]:
          Index = 65
          Value = 0
          Unit = kgm^2
          Description = Jzz5
        Row[67]:
          Index = 66
          Value = 0.394
          Unit = kg
          Description = m6
        Row[68]:
          Index = 67
          Value = 0
          Unit = kgm
          Description = m6*rc6x
        Row[69]:
          Index = 68
          Value = 0
          Unit = kgm
          Description = m6*rc6y
        Row[70]:
          Index = 69
          Value = 0.16745
          Unit = kgm
          Description = m6*rc6z
        Row[71]:
          Index = 70
          Value = 0
          Unit = kgm^2
          Description = m6*rc6x*rc6y
        Row[72]:
          Index = 71
          Value = 0
          Unit = kgm^2
          Description = m6*rc6y*rc6z
        Row[73]:
          Index = 72
          Value = 0
          Unit = kgm^2
          Description = m6*rc6x*rc6z
        Row[74]:
          Index = 73
          Value = 0
          Unit = kgm^2
          Description = m6*rc6x^2
        Row[75]:
          Index = 74
          Value = 0
          Unit = kgm^2
          Description = m6*rc6y^2
        Row[76]:
          Index = 75
          Value = 0.16745
          Unit = kgm^2
          Description = m6*rc6z^2
        Row[77]:
          Index = 76
          Value = 0.038
          Unit = kgm^2
          Description = Jxx6
        Row[78]:
          Index = 77
          Value = 0.038
          Unit = kgm^2
          Description = Jyy6
        Row[79]:
          Index = 78
          Value = 0
          Unit = kgm^2
          Description = Jzz6
        Row[80]:
          Index = 79
          Value = 0.505
          Unit = kg
          Description = m7
        Row[81]:
          Index = 80
          Value = 0
          Unit = kgm
          Description = m7*rc7x
        Row[82]:
          Index = 81
          Value = 0
          Unit = kgm
          Description = m7*rc7y
        Row[83]:
          Index = 82
          Value = 0.133825
          Unit = kgm
          Description = m7*rc7z
        Row[84]:
          Index = 83
          Value = 0
          Unit = kgm^2
          Description = m7*rc7x*rc7y
        Row[85]:
          Index = 84
          Value = 0
          Unit = kgm^2
          Description = m7*rc7y*rc7z
        Row[86]:
          Index = 85
          Value = 0
          Unit = kgm^2
          Description = m7*rc7x*rc7z
        Row[87]:
          Index = 86
          Value = 0
          Unit = kgm^2
          Description = m7*rc7x^2
        Row[88]:
          Index = 87
          Value = 0
          Unit = kgm^2
          Description = m7*rc7y^2
        Row[89]:
          Index = 88
          Value = 0.035463625
          Unit = kgm^2
          Description = m7*rc7z^2
        Row[90]:
          Index = 89
          Value = 0.02385687
          Unit = kgm^2
          Description = Jxx7
        Row[91]:
          Index = 90
          Value = 0.02385687
          Unit = kgm^2
          Description = Jyy7
        Row[92]:
          Index = 91
          Value = 0.000211066
          Unit = kgm^2
          Description = Jzz7
        Row[93]:
          Index = 92
          Value = 0.446
          Unit = kg
          Description = m8
        Row[94]:
          Index = 93
          Value = 0
          Unit = kgm
          Description = m8*rc8x
        Row[95]:
          Index = 94
          Value = 0
          Unit = kgm
          Description = m8*rc8y
        Row[96]:
          Index = 95
          Value = 0.12042
          Unit = kgm
          Description = m8*rc8z
        Row[97]:
          Index = 96
          Value = 0
          Unit = kgm^2
          Description = m8*rc8x*rc8y
        Row[98]:
          Index = 97
          Value = 0
          Unit = kgm^2
          Description = m8*rc8y*rc8z
        Row[99]:
          Index = 98
          Value = 0
          Unit = kgm^2
          Description = m8*rc8x*rc8z
        Row[100]:
          Index = 99
          Value = 0
          Unit = kgm^2
          Description = m8*rc8x^2
        Row[101]:
          Index = 100
          Value = 0
          Unit = kgm^2
          Description = m8*rc8y^2
        Row[102]:
          Index = 101
          Value = 0.0325134
          Unit = kgm^2
          Description = m8*rc8z^2
        Row[103]:
          Index = 102
          Value = 0.019126177
          Unit = kgm^2
          Description = Jxx8
        Row[104]:
          Index = 103
          Value = 0.019126177
          Unit = kgm^2
          Description = Jyy8
        Row[105]:
          Index = 104
          Value = 0.00007511
          Unit = kgm^2
          Description = Jzz8
        Row[106]:
          Index = 105
          Value = 0.505
          Unit = kg
          Description = m9
        Row[107]:
          Index = 106
          Value = 0
          Unit = kgm
          Description = m9*rc9x
        Row[108]:
          Index = 107
          Value = 0
          Unit = kgm
          Description = m9*rc9y
        Row[109]:
          Index = 108
          Value = 0.133825
          Unit = kgm
          Description = m9*rc9z
        Row[110]:
          Index = 109
          Value = 0
          Unit = kgm^2
          Description = m9*rc9x*rc9y
        Row[111]:
          Index = 110
          Value = 0
          Unit = kgm^2
          Description = m9*rc9y*rc9z
        Row[112]:
          Index = 111
          Value = 0
          Unit = kgm^2
          Description = m9*rc9x*rc9z
        Row[113]:
          Index = 112
          Value = 0
          Unit = kgm^2
          Description = m9*rc9x^2
        Row[114]:
          Index = 113
          Value = 0
          Unit = kgm^2
          Description = m9*rc9y^2
        Row[115]:
          Index = 114
          Value = 0.035463625
          Unit = kgm^2
          Description = m9*rc9z^2
        Row[116]:
          Index = 115
          Value = 0.02385687
          Unit = kgm^2
          Description = Jxx9
        Row[117]:
          Index = 116
          Value = 0.02385687
          Unit = kgm^2
          Description = Jyy9
        Row[118]:
          Index = 117
          Value = 0.000213857
          Unit = kgm^2
          Description = Jzz9
        Row[119]:
          Index = 118
          Value = 0.446
          Unit = kg
          Description = m10
        Row[120]:
          Index = 119
          Value = 0
          Unit = kgm
          Description = m10*rc10x
        Row[121]:
          Index = 120
          Value = 0
          Unit = kgm
          Description = m10*rc10y
        Row[122]:
          Index = 121
          Value = 0.12042
          Unit = kgm
          Description = m10*rc10z
        Row[123]:
          Index = 122
          Value = 0
          Unit = kgm^2
          Description = m10*rc10x*rc10y
        Row[124]:
          Index = 123
          Value = 0
          Unit = kgm^2
          Description = m10*rc10y*rc10z
        Row[125]:
          Index = 124
          Value = 0
          Unit = kgm^2
          Description = m10*rc10x*rc10z
        Row[126]:
          Index = 125
          Value = 0
          Unit = kgm^2
          Description = m10*rc10x^2
        Row[127]:
          Index = 126
          Value = 0
          Unit = kgm^2
          Description = m10*rc10y^2
        Row[128]:
          Index = 127
          Value = 0.0325134
          Unit = kgm^2
          Description = m10*rc10z^2
        Row[129]:
          Index = 128
          Value = 0.019126177
          Unit = kgm^2
          Description = Jxx10
        Row[130]:
          Index = 129
          Value = 0.019126177
          Unit = kgm^2
          Description = Jyy10
        Row[131]:
          Index = 130
          Value = 0.0000944
          Unit = kgm^2
          Description = Jzz10
        Row[132]:
          Index = 131
          Value = 1.478
          Unit = kg
          Description = m11
        Row[133]:
          Index = 132
          Value = 0.020692
          Unit = kgm
          Description = m11*rc11x
        Row[134]:
          Index = 133
          Value = 0
          Unit = kgm
          Description = m11*rc11y
        Row[135]:
          Index = 134
          Value = -0.047296
          Unit = kgm
          Description = m11*rc11z
        Row[136]:
          Index = 135
          Value = 0
          Unit = kgm^2
          Description = m11*rc11x*rc11y
        Row[137]:
          Index = 136
          Value = 0
          Unit = kgm^2
          Description = m11*rc11y*rc11z
        Row[138]:
          Index = 137
          Value = -0.000662144
          Unit = kgm^2
          Description = m11*rc11x*rc11z
        Row[139]:
          Index = 138
          Value = 0.000289688
          Unit = kgm^2
          Description = m11*rc11x^2
        Row[140]:
          Index = 139
          Value = 0
          Unit = kgm^2
          Description = m11*rc11y^2
        Row[141]:
          Index = 140
          Value = 0.001513472
          Unit = kgm^2
          Description = m11*rc11z^2
        Row[142]:
          Index = 141
          Value = 0
          Unit = kgm^2
          Description = Jxx11
        Row[143]:
          Index = 142
          Value = 0
          Unit = kgm^2
          Description = Jyy11
        Row[144]:
          Index = 143
          Value = 0
          Unit = kgm^2
          Description = Jzz11
        Row[145]:
          Index = 144
          Value = 0
          Unit = kg
          Description = m12
        Row[146]:
          Index = 145
          Value = 0
          Unit = kgm
          Description = m12*rc12x
        Row[147]:
          Index = 146
          Value = 0
          Unit = kgm
          Description = m12*rc12y
        Row[148]:
          Index = 147
          Value = 0
          Unit = kgm
          Description = m12*rc12z
        Row[149]:
          Index = 148
          Value = 0
          Unit = kgm^2
          Description = m12*rc12x*rc12y
        Row[150]:
          Index = 149
          Value = 0
          Unit = kgm^2
          Description = m12*rc12y*rc12z
        Row[151]:
          Index = 150
          Value = 0
          Unit = kgm^2
          Description = m12*rc12x*rc12z
        Row[152]:
          Index = 151
          Value = 0
          Unit = kgm^2
          Description = m12*rc12x^2
        Row[153]:
          Index = 152
          Value = 0
          Unit = kgm^2
          Description = m12*rc12y^2
        Row[154]:
          Index = 153
          Value = 0
          Unit = kgm^2
          Description = m12*rc12z^2
        Row[155]:
          Index = 154
          Value = 0
          Unit = kgm^2
          Description = Jxx12
        Row[156]:
          Index = 155
          Value = 0
          Unit = kgm^2
          Description = Jyy12
        Row[157]:
          Index = 156
          Value = 0.00039
          Unit = kgm^2
          Description = Jzz12
        Row[158]:
          Index = 157
          Value = 0.23
          Unit = kg
          Description = m13
        Row[159]:
          Index = 158
          Value = 0
          Unit = kgm
          Description = m13*rc13x
        Row[160]:
          Index = 159
          Value = 0.006785
          Unit = kgm
          Description = m13*rc13y
        Row[161]:
          Index = 160
          Value = 0
          Unit = kgm
          Description = m13*rc13z
        Row[162]:
          Index = 161
          Value = 0
          Unit = kgm^2
          Description = m13*rc13x*rc13y
        Row[163]:
          Index = 162
          Value = 0
          Unit = kgm^2
          Description = m13*rc13y*rc13z
        Row[164]:
          Index = 163
          Value = 0
          Unit = kgm^2
          Description = m13*rc13x*rc13z
        Row[165]:
          Index = 164
          Value = 0
          Unit = kgm^2
          Description = m13*rc13x^2
        Row[166]:
          Index = 165
          Value = 0.0002001575
          Unit = kgm^2
          Description = m13*rc13y^2
        Row[167]:
          Index = 166
          Value = 0
          Unit = kgm^2
          Description = m13*rc13z^2
        Row[168]:
          Index = 167
          Value = 0.00045
          Unit = kgm^2
          Description = Jxx13
        Row[169]:
          Index = 168
          Value = 0
          Unit = kgm^2
          Description = Jyy13
        Row[170]:
          Index = 169
          Value = 0.00081
          Unit = kgm^2
          Description = Jzz13
        Row[171]:
          Index = 183
          Value = 0.000393
          Unit = kgm^2
          Description = JDrive1
        Row[172]:
          Index = 184
          Value = 0.000393
          Unit = kgm^2
          Description = JDrive2
        Row[173]:
          Index = 185
          Value = 0.000393
          Unit = kgm^2
          Description = JDrive3
        Row[174]:
          Index = 186
          Value = 0.000092
          Unit = kgm^2
          Description = JDrive4
        Row[175]:
          Index = 187
          Value = 0.000092
          Unit = kgm^2
          Description = JDrive5
        Row[176]:
          Index = 188
          Value = 0.249554950768092
          Unit = Nms
          Description = dV1
        Row[177]:
          Index = 189
          Value = 0.249554950768092
          Unit = Nms
          Description = dV2
        Row[178]:
          Index = 190
          Value = 0.249554950768092
          Unit = Nms
          Description = dV3
        Row[179]:
          Index = 191
          Value = 1.59154943091895E-02
          Unit = Nms
          Description = dV4
        Row[180]:
          Index = 192
          Value = 1.59154943091895E-02
          Unit = Nms
          Description = dV5
        Row[181]:
          Index = 193
          Value = 6.16
          Unit = Nm
          Description = dC1
        Row[182]:
          Index = 194
          Value = 6.16
          Unit = Nm
          Description = dC2
        Row[183]:
          Index = 195
          Value = 6.16
          Unit = Nm
          Description = dC3
        Row[184]:
          Index = 196
          Value = 1
          Unit = Nm
          Description = dC4
        Row[185]:
          Index = 197
          Value = 1
          Unit = Nm
          Description = dC5
      DynamicLimits = DynParTables
        GearboxLimitsTableRef
        CrossSectionLimitsTableRef
      InternalDynamicLimits = Used
        TypeIsReadOnly = 1
        Type = D5-1100-S026-R100
        GearboxLimits:
          Row[1]:
            Index = 0
            Value = 3
            Unit = 
            Description = Type of robot dyn par model
          Row[2]:
            Index = 1
            Value = 85
            Unit = Nm
            Description = Gearbox Drive 1
          Row[3]:
            Index = 2
            Value = 85
            Unit = Nm
            Description = Gearbox Drive 2
          Row[4]:
            Index = 3
            Value = 85
            Unit = Nm
            Description = Gearbox Drive 3
          Row[5]:
            Index = 4
            Value = 3.5
            Unit = Nm
            Description = Gearbox Drive 4
          Row[6]:
            Index = 5
            Value = 3.5
            Unit = Nm
            Description = Gearbox Drive 5
        CrossSectionLimits:
          Row[1]:
            Index = 0
            Value = 3
            Unit = Variant
            Description = 
          Row[2]:
            Index = 1
            Value = 100
            Unit = N
            Description = 
          Row[3]:
            Index = 2
            Value = 100
            Unit = N
            Description = 
          Row[4]:
            Index = 3
            Value = 100
            Unit = N
            Description = 
          Row[5]:
            Index = 4
            Value = 4
            Unit = Nm
            Description = 
          Row[6]:
            Index = 5
            Value = 10
            Unit = Nm
            Description = 
          Row[7]:
            Index = 6
            Value = 10
            Unit = Nm
            Description = 
          Row[8]:
            Index = 7
            Value = 100
            Unit = N
            Description = 
          Row[9]:
            Index = 8
            Value = 100
            Unit = N
            Description = 
          Row[10]:
            Index = 9
            Value = 100
            Unit = N
            Description = 
          Row[11]:
            Index = 10
            Value = 10
            Unit = N
            Description = 
          Row[12]:
            Index = 11
            Value = 10
            Unit = N
            Description = 
          Row[13]:
            Index = 12
            Value = 5
            Unit = N
            Description = 
          Row[14]:
            Index = 13
            Value = 225
            Unit = N
            Description = 
          Row[15]:
            Index = 14
            Value = 225
            Unit = N
            Description = 
          Row[16]:
            Index = 15
            Value = 225
            Unit = N
            Description = 
          Row[17]:
            Index = 16
            Value = 225
            Unit = N
            Description = 
          Row[18]:
            Index = 17
            Value = 225
            Unit = N
            Description = 
          Row[19]:
            Index = 18
            Value = 225
            Unit = N
            Description = 
      LoadDependentJerkLimitsIsReadOnly = 0
      LoadDependentJerkLimits = NotUsed
      CouplingsIsInvisible = 0
      Couplings:
        LinearCoupling[1]:
          SourceAxisIsReadOnly = 1
          SourceAxis = 4
          SourceAxisUnitsIsReadOnly = 1
          SourceAxisUnits = 2
          TargetJointAxisIsReadOnly = 1
          TargetJointAxis = 4
          TargetJointAxisUnitsIsReadOnly = 1
          TargetJointAxisUnits = 1
        LinearCoupling[2]:
          SourceAxisIsReadOnly = 1
          SourceAxis = 5
          SourceAxisUnitsIsReadOnly = 1
          SourceAxisUnits = 2
          TargetJointAxisIsReadOnly = 1
          TargetJointAxis = 5
          TargetJointAxisUnitsIsReadOnly = 1
          TargetJointAxisUnits = 1
        LinearCoupling[3]:
          SourceAxisIsReadOnly = 1
          SourceAxis = 4
          SourceAxisUnitsIsReadOnly = 1
          SourceAxisUnits = -4
          TargetJointAxisIsReadOnly = 1
          TargetJointAxis = 5
          TargetJointAxisUnitsIsReadOnly = 1
          TargetJointAxisUnits = 1
      JointAxesPositionLimits:
        JointAxisIsReadOnly = 0
        JointAxis[1] = UseAxisLimits
        JointAxis[2] = UseAxisLimits
        JointAxis[3] = UseAxisLimits
        JointAxis[4] = UseAxisLimits
        JointAxis[5] = UseAxisLimits
      WorkingRangeIsReadOnly = 0
      WorkingRange = Standard
        BaseToTopIsReadOnly = 0
        BaseToTop = 706
        TopHeightIsReadOnly = 0
        TopHeight = 40
        MiddleHeightIsReadOnly = 0
        MiddleHeight = 210
        BottomHeightIsReadOnly = 0
        BottomHeight = 150
        TopRadiusIsReadOnly = 0
        TopRadius = 517
        MiddleRadiusIsReadOnly = 0
        MiddleRadius = 551
        BottomRadiusIsReadOnly = 0
        BottomRadius = 335
```

### Config_9.axesgroupfeature - 5APC3100_KBU3_000/mappMotion/Codian_D5r1100R_1/Config_9.axesgroupfeature
```
Element Feature_Programs_D5r1100R_1 (Type=axesgroupfeature)
  Type = Program
    ModalDataBehaviour = UseAxesGroupSettings
    InitialSettings:
      InterpolationTypes = LinearRapid
      PositionCoordinates = Absolute
      CircleCoordinates = Relative
      JACS_ACSProgramming = JACS
      ContourConnection = Inactive
      AccuracyHoldDelays = User defined
        UserAxesDelay = 0.06
        UserDelay = 0.0
      ProgrammingUnits = UseAxesGroupSettings
      Feedrates:
        FeedPath = Standard
        FeedCharacteristic = StandardCharacteristic
        FeedType = Feedrate
        FeedReduction = Inactive
        FeedrateValue = 0.0
        InverseFeedrateValue = 0.0
        FeedratePerRevValue = 0.0
    DefaultLanguage = BRGCode
    Location = Default
      FileDevice = CNC_PrgDir
    ProgramElements:
      PVs:
        PV[1]:
          PvName = ::APP_Robot1:MaxPickPosX
          Advanced:
            Alias = MaxPickPosX
            Synchronization = Ip
            Reference = No
        PV[2]:
          PvName = ::APP_Robot1:MinPickPosX
          Advanced:
            Alias = MinPickPosX
            Synchronization = Ip
            Reference = No
        PV[3]:
          PvName = ::APP_Robot1:PickTrackingObject
          Advanced:
            Alias = PickTrackingObject
            Synchronization = Ip
            Reference = No
        PV[4]:
          PvName = ::APP_Robot1:MinPlacePosX
          Advanced:
            Alias = MinPlacePosX
            Synchronization = Ip
            Reference = No
        PV[5]:
          PvName = ::APP_Robot1:MaxPlacePosX
          Advanced:
            Alias = MaxPlacePosX
            Synchronization = Ip
            Reference = No
        PV[6]:
          PvName = ::APP_Robot1:PlaceTrackingObject
          Advanced:
            Alias = PlaceTrackingObject
            Synchronization = Ip
            Reference = No
        PV[7]:
          PvName = ::ControlPanel.Input.Conveyor2.VelocityProduction
          Advanced:
            Alias = BeltSpeed
            Synchronization = Ip
            Reference = No
```

### ComRobot.axesgroupfeature - 5APC3100_KBU3_000/mappMotion/ComRobot.axesgroupfeature
```
Element Feature_TrackingRobot (Type=axesgroupfeature)
  Type = Tracking
    MotionBehaviour:
      OutOfWorkspaceSynchronisation:
        Clearance = 10
Element Feature_MFunctions (Type=axesgroupfeature)
  Type = MFunctions
    MFunction[1]:
      IndexType:
        Index = 8
      Blocking = Disabled
      InSimulation = Set
      PvMapping = ::APP_Robot1:M8
    MFunction[2]:
      IndexType:
        Index = 9
      Blocking = Disabled
      InSimulation = Set
      PvMapping = ::APP_Robot1:M9
    MFunction[3]:
      IndexType:
        Index = 16
      InSimulation = Set
      PvMapping = ::APP_Robot1:M16
    MFunction[4]:
      IndexType:
        Index = 17
      InSimulation = Set
      PvMapping = ::APP_Robot1:M17
    MFunction[5]:
      IndexType:
        Index = 20
      PvMapping = ::APP_Robot1:M20
    MFunction[6]:
      IndexType:
        Index = 21
      PvMapping = ::APP_Robot1:M21
Element Feature_InterpreterLog (Type=axesgroupfeature)
  Type = MotionPacketLog
Element Feature_Monitoring (Type=axesgroupfeature)
  Type = MonitoringElements
    CombinedElements:
      BasicMonitor = ::APP_Robot1:BasicMonitor
    SingleElements:
      SingleElement[1] = Interpreter
        IpMonitor = ::APP_Robot1:IPMonitor
Element Feature_PathDefRobot (Type=axesgroupfeature)
  Type = PathDefinitions
    PathDefinition[1]:
      Type:
        CalculatedIn = PCS
Element Feature_FrameHierachy (Type=axesgroupfeature)
  Type = FrameHierarchy
    FrameHierarchy = Custom
      FramePropertyMapping:
        BCS = RobotBase
      MCS:
        Frame[1]:
          Name = RobotBase
          Type:
            Translation:
              Z = 1000
        Frame[2]:
          Name = UserFrame1
Element Feature_WorkspaceMonitoring (Type=axesgroupfeature)
  Type = WorkspaceMonitoring
    WorkspaceRef = Workspace_1
Element Feature_Signaling (Type=axesgroupfeature)
  Type = Signaling
    Prediction:
      Time = Used
        Time = 0.045
    Signals:
      UnconfiguredSignals:
        MissedSignalBehaviour = DelayedOutputAndWarning
      Signal[1]:
        Name = Sig8
        Action:
          Index = 8
        ReactionTime = Used
        MissedSignalBehaviour = DelayedOutputAndWarning
      Signal[2]:
        Name = Sig9
        Action:
          Index = 9
        ReactionTime = Used
        MissedSignalBehaviour = DelayedOutputAndWarning
      Signal[3]:
        Name = Sig16
        Action:
          Index = 16
        MissedSignalBehaviour = DelayedOutputAndWarning
      Signal[4]:
        Name = Sig17
        Action:
          Index = 17
        MissedSignalBehaviour = DelayedOutputAndWarning
Element Feature_Tool (Type=axesgroupfeature)
  Type = Tools
    Tools:
      ToolTable = ToolTable_1
      Index = 3
```

### AxisAx_1.axis - 5APC3100_KBU3_000/mappMotion/Conveyor/AxisAx_1.axis
```
Element AxConveyorOut (Type=axis)
  BaseTypeIsReadOnly = 0
  BaseType = LinearPeriodic
    MeasurementUnit = 5066068
    MeasurementResolutionIsReadOnly = 0
    MeasurementResolution = 0.01
    CountDirectionIsReadOnly = 0
    CountDirection = Standard
    PeriodSettings:
      Period = 100000.0
  MovementLimitsIsReadOnly = 0
  MovementLimits = Internal
    Position:
      LowerLimitMin = -1.79769313486231E308
      UpperLimitMax = 1.79769313486231E308
      LowerLimit = -8388608.0
      UpperLimit = 8388607.0
    VelocityIsReadOnly = 0
    Velocity:
      VelocityMax = 3.4E38
      Velocity = 1000.0
    AccelerationIsReadOnly = 0
    Acceleration:
      AccelerationMax = 3.4E38
      Acceleration = 5000.0
    DecelerationIsReadOnly = 0
    Deceleration:
      DecelerationMax = 3.4E38
      Deceleration = 5000.0
  Alarms = None
Element AxConveyorIn (Type=axis)
  BaseTypeIsReadOnly = 0
  BaseType = LinearPeriodic
    MeasurementUnit = 5066068
    MeasurementResolutionIsReadOnly = 0
    MeasurementResolution = 0.01
    CountDirectionIsReadOnly = 0
    CountDirection = Standard
    PeriodSettings:
      Period = 100000.0
  MovementLimitsIsReadOnly = 0
  MovementLimits = Internal
    Position:
      LowerLimitMin = -1.79769313486231E308
      UpperLimitMax = 1.79769313486231E308
      LowerLimit = -8388608.0
      UpperLimit = 8388607.0
    VelocityIsReadOnly = 0
    Velocity:
      VelocityMax = 3.4E38
      Velocity = 1000.0
    AccelerationIsReadOnly = 0
    Acceleration:
      AccelerationMax = 3.4E38
      Acceleration = 5000.0
    DecelerationIsReadOnly = 0
    Deceleration:
      DecelerationMax = 3.4E38
      Deceleration = 5000.0
  Alarms = None
```

### Config_1.trackingpath - 5APC3100_KBU3_000/mappMotion/Conveyor/Config_1.trackingpath
```
Element gTrackingPathConveyorOut (Type=trackingpath)  // Tracking Path with moving objects
  Type = Linear
    MotionSource = Axis
      AxisRef = AxConveyorOut
      AxisUsage:
        CommandConsideration = SupportBasicCommands
  SceneViewerObject = Used
  Alarms = None
Element gTrackingPathConveyorIn (Type=trackingpath)  // Tracking Path with moving objects
  Type = Linear
    MotionSource = Axis
      AxisRef = AxConveyorIn
  SceneViewerObject = Used
  Alarms = None
```

### Config_3.axisfeature - 5APC3100_KBU3_000/mappMotion/Conveyor/Config_3.axisfeature
```
Element AxProfGenJerkLim (Type=axisfeature)
  Type = ProfGen
    JerkFilter = JerkLimited
```

## Logical view

Binary libraries used (declarations not repeated): operator, runtime, astime, AsIecCon, standard, AsBrStr, sys_lib, AsArSdm, brsystem, FileIO, AsIODiag, DataObj, AsArProf, AsMem, AsIOAcc, AsEPL, ASMcDcs, AsBrMath, visapi, ArTextSys, AsSem, AsZip, AcpInvLib, MpRecipe, MpUserX, MpFile, MpAlarmX, MpCom, CoTrace, MpServer, McBase, MpBase, MpAxis, McAcpAx, McPathGen, McPureVAx, McAxGroup, McAxis, McProgInt, McTrkPath, McDS402Ax, MpRobotics, MpCnc, MpTool 6.2.0

### MachineInterface.var
```iecst
(*Defines*)
VAR CONSTANT
	MAX_TRACKING_FRAMES : USINT := 40; (*Number of supported objects on the tracking frame*)
	NUM_DEVICES : DINT := 2; (*Number of devices (Robots + Axis)*)
END_VAR
(*Stores the Devices Conveyor & Robot 1*)
VAR CONSTANT
	DEVICES_ARRAY : INT := NUM_DEVICES-1; (*Size of devices array*)
END_VAR
(*Internal states*)
VAR
	ControlPanel : ControlPanelType := (Input:=(Start:=FALSE,Reset:=FALSE,Conveyor1:=(YShift:=0,VelocityProduction:=20,ProductGap:=100,DeletePosition:=800),Conveyor2:=(YShift:=0,VelocityProduction:=200,IndexingDistance:=400,ProductGap:=450,DeletePosition:=2000),ProgramRobot1:='Track.st')); (*Machine interface (inputs/outputs)*)
END_VAR
```

### MachineInterface.typ
```iecst
TYPE
	ConveyorSettings : 	STRUCT  (*Command Buttons*)
		YShift : LREAL; (*Min Y Pos in Random mode*)
		VelocityProduction : REAL; (*Velocity for production [ppm]*)
		IndexingDistance : REAL; (*Indexing distance [mm]*)
		ProductGap : REAL; (*Length of the product [mm]*)
		DeletePosition : REAL; (*Position where objects are deleted*)
	END_STRUCT;
	ControlPanelInputs : 	STRUCT  (*Command Buttons*)
		Start : BOOL; (*Run Applicaion*)
		Reset : BOOL; (*Reset Error states*)
		Conveyor1 : ConveyorSettings; (*Buttons *)
		Conveyor2 : ConveyorSettings; (*Buttons *)
		ProgramRobot1 : STRING[32]; (*Program name for robot 1*)
	END_STRUCT;
	ControlPanelType : 	STRUCT  (*Control Panel*)
		Input : ControlPanelInputs; (*Buttons *)
	END_STRUCT;
END_TYPE

(*Device Interface*)
(*
Enumerators for State Machnie (used at Conveyor and Robot)*)

TYPE
	DeviceStatesListEnum :
		( (*State of the robot / axis*)
		STATE_WAIT, (*Standby*)
		STATE_INIT, (*Initialization*)
		STATE_PRODUCTION, (*Production*)
		STATE_ERROR, (*Emenrgency*)
		STATE_RESET (*Reset*)
		);
END_TYPE

(*
Product positions for SceneViewer*)

TYPE
	ProdPosType : 	STRUCT  (*Visu position for Scene Viewer*)
		Full : BOOL; (*Display object*)
		Valid : BOOL; (*Display object*)
		Element1 : BOOL; (*Display object*)
		Element2 : BOOL; (*Display object*)
		Empty : BOOL; (*Display object*)
		PositionX : REAL; (*Pos X*)
		PositionY : REAL; (*Pos Y*)
		PositionZ : REAL; (*Pos Z*)
		Material : UDINT; (*Material Color to show Tracking*)
	END_STRUCT;
END_TYPE
```


### Package Logical/Conveyor - Device: 1 axis positioner

### Program Logical/Conveyor/APP_ConveyorIn (IEC) - Motion Belt

#### Variables.var - Local variables
```iecst
(*
MpAxisBasic function blocks used for Conveyor Handling*)
VAR
	MpAxConveyor : MpAxisBasic;
	AxParConveyor : MpAxisBasicParType;
	McCfgAxConveyor : McCfgAxBaseTypType;
	TrackLinkConveyor : UDINT;
	AxGroupLink : UDINT;
END_VAR
(*
MpAxisBasicConfig function blocks*)
VAR
	MoveAbsoluteLastPosition : LREAL := 0;
	LastProductPosition : LREAL := 0;
	State : DeviceStatesListEnum; (*Statemachine of conveyor*)
	i : INT := 0; (*Loop counter*)
END_VAR
(*
Tracking function*)
VAR
	MC_BR_TrackingFrameCreate_0 : MC_BR_TrackingFrameCreate;
	MC_BR_TrackingPathGetFrames_0 : MC_BR_TrackingPathGetFrames;
	MC_MoveVelocity_0 : MC_MoveVelocity;
	MC_BR_TrackingPathReset_0 : MC_BR_TrackingPathReset;
	MC_BR_TrackingPathReadStatus_0 : MC_BR_TrackingPathReadStatus;
	MC_BR_TrackingPathReadInfo_0 : MC_BR_TrackingPathReadInfo;
	MC_Stop_0 : MC_Stop;
	MC_MoveAdditive_0 : MC_MoveAdditive;
	MC_BR_TrackingFrameDelete_0 : MC_BR_TrackingFrameDelete;
	Products : ARRAY[0..MAX_TRACKING_FRAMES] OF McTrkFrmInfoType; (*Memory holding all tracking frames (Get Frames)*)
	ProductDetails : ARRAY[0..MAX_TRACKING_FRAMES] OF ProductDetailsType; (*Additional Attribute memory for the tracking frames*)
	ParkPosition : LREAL := 0; (*Fixed Belt - Workaround *)
	ProdDetails : REFERENCE TO ProductDetailsType; (*Scene Viewer*)
	ConvSettings : REFERENCE TO ConveyorSettings;
END_VAR
(*
Product positions (Variable for Scene Viewer)*)
VAR
	ProductsPosition : ARRAY[0..MAX_TRACKING_FRAMES] OF ProdPosType; (*Scene Viewer Data*)
	AxWithCommandConsideration : BOOL;
END_VAR
```

#### Init.st - Init code
```iecst
PROGRAM _INIT

	TrackLinkConveyor := ADR(gTrackingPathConveyorIn);
	AxGroupLink := ADR(AxConveyorIn);
	ConvSettings ACCESS ADR(ControlPanel.Input.Conveyor1);
	AxWithCommandConsideration := FALSE;

	initConveyor;

END_PROGRAM
```

#### Cyclic.st - Cyclic code
```iecst
PROGRAM _CYCLIC

	CASE State OF

		/////////////////////////////////////////////////////////////////////////////
		STATE_WAIT:
		/////////////////////////////////////////////////////////////////////////////
			IF  ControlPanel.Input.Start THEN
				State := 	STATE_INIT;
			END_IF

		/////////////////////////////////////////////////////////////////////////////
		STATE_INIT:
		////////////////////////////////////////////////////////////////////////////

			IF MpAxConveyor.CommandBusy THEN
				// wait
			ELSIF NOT(MpAxConveyor.Active) THEN
				MpAxConveyor.Enable := TRUE;

			ELSIF MpAxConveyor.Error THEN
				MpAxConveyor.ErrorReset := TRUE;

			ELSIF NOT(MpAxConveyor.PowerOn) THEN
				MpAxConveyor.Power := TRUE;

			ELSIF NOT(MpAxConveyor.IsHomed) THEN
				AxParConveyor.Homing.Mode := mcHOMING_DIRECT;
				AxParConveyor.Homing.Position := 0;
				MpAxConveyor.Home := TRUE;

			ELSIF MpAxConveyor.Info.CommunicationReady THEN
				LastProductPosition := MpAxConveyor.Position - ConvSettings.ProductGap;
				brsmemset(ADR(Products), 0, SIZEOF(Products));
				State := STATE_PRODUCTION;
			END_IF

		//////////////////////////////////////// Frame Handling! + Stat Machine Conveyor///////////////////////////////////////
		STATE_PRODUCTION:
		///////////////////////////////////////////////////////////////////////////////

			// Frame Handling
			MC_BR_TrackingPathGetFrames_0.Execute := NOT(MC_BR_TrackingPathGetFrames_0.Done);
			IF MC_BR_TrackingPathGetFrames_0.Done AND NOT MC_BR_TrackingPathGetFrames_0.Busy AND NOT(MC_BR_TrackingFrameDelete_0.Execute) AND NOT(MC_BR_TrackingFrameCreate_0.Execute) THEN

				// Update the Data of the products stored in the product buffer
				updateProductData;
				// Find & Delete Products, which are out of scope
				deleteOutOfScopeProducts;
				IF  NOT (MC_BR_TrackingFrameDelete_0.Execute)																																	AND
					((MpAxConveyor.Position >= LastProductPosition + ConvSettings.ProductGap) 																							OR
					(MpAxConveyor.Position < LastProductPosition AND (LastProductPosition + ConvSettings.ProductGap >= McCfgAxConveyor.BaseType.LinearPeriodic.PeriodSettings.Period))) 	THEN

					addNewObjects;
				END_IF

			END_IF

			IF MC_MoveAdditive_0.Error OR MC_MoveVelocity_0.Error OR MC_Stop_0.Error OR MpAxConveyor.Error OR MC_BR_TrackingPathReadStatus_0.TrackingPathErrorStop THEN
				State := STATE_ERROR;
				MpAxConveyor.Power := FALSE;

			ELSIF NOT(ControlPanel.Input.Start) THEN
				IF MpAxConveyor.MoveActive THEN
					MC_Stop_0.Execute := NOT MC_Stop_0.Busy;
				ELSIF MpAxConveyor.PowerOn AND NOT MC_Stop_0.Busy THEN
					MpAxConveyor.Power := FALSE;
				ELSE
					State := STATE_WAIT;
				END_IF
			ELSE
				applyBeltMovement;
			END_IF

		///////////////////////////////////////////////////////////////////////////////
		STATE_ERROR:
		///////////////////////////////////////////////////////////////////////////////
			MpAxConveyor.Power := FALSE;
			IF MpAxConveyor.Error OR MpAxConveyor.CommandBusy OR MC_BR_TrackingPathReset_0.Busy OR MC_BR_TrackingPathReset_0.Error OR MC_BR_TrackingPathReadStatus_0.TrackingPathErrorStop THEN
				IF ControlPanel.Input.Reset THEN
					MpAxConveyor.ErrorReset := TRUE;
					MC_BR_TrackingPathReset_0.Execute := TRUE;

					brsmemset(ADR(Products), 0, SIZEOF(Products));
					brsmemset(ADR(ProductDetails), 0, SIZEOF(ProductDetails));
				END_IF
			ELSE
				State := STATE_WAIT;
			END_IF

	END_CASE

	(* *************************************************************************************************************************** *)
	(* *************************************************************************************************************************** *)
	(* *************************************************************************************************************************** *)

	// Function blocks call
	MpAxConveyor(MpLink := AxGroupLink,	Parameters := ADR(AxParConveyor));

	// movement fubs
	MC_MoveAdditive_0(Axis := AxGroupLink);
	MC_MoveAdditive_1(Axis := AxGroupLink);
	MC_MoveVelocity_0(Axis := AxGroupLink);
	MC_Stop_0(Axis := AxGroupLink);

	// Tracking commands
	MC_BR_TrackingFrameCreate_0(TrackingPath := TrackLinkConveyor);
	MC_BR_TrackingPathGetFrames_0(TrackingPath := TrackLinkConveyor);
	MC_BR_TrackingFrameDelete_0(TrackingPath := TrackLinkConveyor);
	MC_BR_TrackingPathReset_0(TrackingPath := TrackLinkConveyor);
	MC_BR_TrackingPathReadStatus_0(TrackingPath := TrackLinkConveyor);

	// Update Scene Viewer positions
	updateSceneViewerPositions;

	(* *************************************************************************************************************************** *)
	(*                                                    RESET PARAMETER 														   *)
	(* *************************************************************************************************************************** *)

	resetFUBs;

END_PROGRAM
```
